// TwinCAT 3 PLC project TwinCAT3_Numpad_Keypad
// ProgramVersion: 3.1.4023.0
// libraries:
//   Tc2_Standard, * (Beckhoff Automation GmbH)
//   Tc2_System, * (Beckhoff Automation GmbH)
//   Tc3_Module, * (Beckhoff Automation GmbH)
//   VisuDialogs, * (System)
// project tree:
//   / GlobalTextList.TcGTLO, PlcTask.TcTTO, Visualization Manager.TcVMO (not stored), VISU_TASK.TcTTO
//   GVLs/ GVL.TcGVL
//   POUs/ MAIN.TcPOU
//   VISUs/Keyboard/ DialogCheckInit.TcPOU, DialogCheckInitForExponential.TcPOU, Dialog_Constants.TcGVL, Dialog_FormatTypes.TcDUT, Dialog_Variables_Exp.TcGVL, Keypad.TcVIS, KeypadLayout.TcVIS, Keypad_Original.TcVIS, Numpad.TcVIS, NumpadExtended.TcVIS, Numpad_Original.TcVIS, VisuDlg_CheckedAppend.TcPOU, VisuDlg_CheckedClear.TcPOU, VisuDlg_CheckedExpFloatFormatSwitch.TcPOU, VisuDlg_GetPasswordString.TcPOU, VisuDlg_ProcessBack.TcPOU, VisuDlg_ProcessChangeNumberFormat.TcPOU, VisuDlg_ProcessChangeSign.TcPOU, VisuDlg_ProcessChangeSignExtended.TcPOU, VisuDlg_ProcessChar.TcPOU, VisuDlg_ProcessCharWithInit.TcPOU, VisuDlg_ProcessClear.TcPOU, VisuDlg_ProcessExp.TcPOU, VisuDlg_ProcessExpFloatFormatSwitch.TcPOU
//   VISUs/ vMain.TcVIS

CONFIGURATION TwinCAT3_Numpad_Keypad
    RESOURCE PLC ON TwinCAT3
        TASK PlcTask(INTERVAL := T#10ms, PRIORITY := 20);
        TASK VISU_TASK(INTERVAL := T#1ms, PRIORITY := 30);
        PROGRAM MAIN WITH PlcTask : MAIN;
        PROGRAM VisuElems_Visu_Prg WITH VISU_TASK : VisuElems.Visu_Prg;
    END_RESOURCE
END_CONFIGURATION

// ---- VISUs/Keyboard/Dialog_FormatTypes.TcDUT
{attribute 'qualified_only'}
TYPE Dialog_FormatTypes :
(
	DECIMAL := 0,
	HEX
);
END_TYPE

// ---- GVLs/GVL.TcGVL
VAR_GLOBAL
  gsPadTitle: STRING;
END_VAR

// ---- VISUs/Keyboard/Dialog_Constants.TcGVL
{attribute 'explicit-init-exit-handling' := 'visu'}
{attribute 'qualified_only'}
VAR_GLOBAL CONSTANT
	PASSWORD_CHAR : STRING(1) := '*';
END_VAR
VAR_GLOBAL
	stTabl: INT;
END_VAR

// ---- VISUs/Keyboard/Dialog_Variables_Exp.TcGVL
{attribute 'explicit-init-exit-handling' := 'visu'}
{attribute: 'global_init_slot' := '150000'}
VAR_GLOBAL
	// Value contains e (exp was pressed)
	g_XExp : BOOL;
END_VAR

// ---- POUs/MAIN.TcPOU
PROGRAM MAIN
VAR
  nTest: INT;
  sTest: STRING;
END_VAR

END_PROGRAM

// ---- VISUs/Keyboard/DialogCheckInit.TcPOU
FUNCTION DialogCheckInit : BOOL
VAR_IN_OUT
	stValue : STRING;
	stOutput : STRING;
	bInit : BOOL;
END_VAR
VAR
END_VAR

IF bInit THEN
	stValue := ''; 
	stOutput := '';
	g_XExp := FALSE;
	// g_Format is reset on close, not on init
	bInit := FALSE;
END_IF

END_FUNCTION

// ---- VISUs/Keyboard/DialogCheckInitForExponential.TcPOU
// On opening of the NumpadExtended, we have to check the display value.
// It can be displayed in exponential notation.
// New function used with the VisuDlg_Process.. functions
FUNCTION DialogCheckInitForExponential : BOOL
VAR_IN_OUT	
	bInit : BOOL;
END_VAR
VAR_INPUT
	stValue : STRING;
END_VAR

// Starting with V3.5.9.0 the value will not be reset, after the first 
// action. Because of the new usage of the textfield with caret and selection.
IF bInit THEN
	bInit := FALSE;
	g_XExp := FALSE;
	
	IF 0 < LEN(stValue) THEN
		// value contains the 'e' character: set flag g_XExp 
		IF FIND(stValue, 'e') > 0 THEN
			g_XExp := TRUE;
		END_IF
	END_IF
	
END_IF

END_FUNCTION

// ---- VISUs/Keyboard/VisuDlg_CheckedAppend.TcPOU
FUNCTION VisuDlg_CheckedAppend : BOOL
VAR_IN_OUT
	stOutputValue : STRING;
	stVariableValue : STRING;
	bInit : BOOL;
END_VAR
VAR_INPUT
	bPassword : BOOL;
	cToAppend : STRING(1);
END_VAR

DialogCheckInit(stVariableValue, stOutputValue, bInit);

stVariableValue := CONCAT(stVariableValue, cToAppend);
IF bPassword THEN
	stOutputValue := CONCAT(stOutputValue, Dialog_Constants.PASSWORD_CHAR);
ELSE
	stOutputValue := stVariableValue;
END_IF

END_FUNCTION

// ---- VISUs/Keyboard/VisuDlg_CheckedClear.TcPOU
// clear for the Numpad, not NumpadBasic
FUNCTION VisuDlg_CheckedClear : Bool
VAR_IN_OUT
	stOutputValue : STRING;
	stVariableValue : STRING;
	flags : DWORD;
END_VAR
VAR
END_VAR

// because of integrated visu, put into a function.
// reason: unknown g_XExp
stVariableValue := '';
stOutputValue := '';
g_XExp := FALSE;
flags := flags AND NOT SINT_TO_DWORD(16#0008);
flags := flags AND NOT SINT_TO_DWORD(16#0010);

END_FUNCTION

// ---- VISUs/Keyboard/VisuDlg_CheckedExpFloatFormatSwitch.TcPOU
// switches the format of the displayed value
// between exponential and float / decimal value
FUNCTION VisuDlg_CheckedExpFloatFormatSwitch : BOOL
VAR_IN_OUT
	stOutputValue : STRING;
	stVariableValue : STRING;
END_VAR
VAR_INPUT
	bPassword: BOOL;
END_VAR
VAR
	// no need to initialize the global flag for exp
	bInitExp : BOOL := FALSE;
	// just dummies, not needed here
	iCaretPosition		: INT;
	iSelectionStart		: INT;
	iSelectionEnd		: INT;
END_VAR

//dont call DialogCheckInit here

VisuDlg_ProcessExpFloatFormatSwitch(stOutputValue, stVariableValue, iCaretPosition, iSelectionStart, iSelectionEnd, bInitExp, bPassword);

END_FUNCTION

// ---- VISUs/Keyboard/VisuDlg_ProcessExpFloatFormatSwitch.TcPOU
/// switches the format of the displayed value
/// between exponential and float / decimal value
/// and changes caret position and selection
FUNCTION VisuDlg_ProcessExpFloatFormatSwitch : BOOL
VAR_IN_OUT
	stOutputValue : STRING;
	stVariableValue : STRING;
	/// The current position of the caret. Either within the text or at the end of the text
	iCaretPosition		: INT;
	/// The start of the selected text (1-relative)
	iSelectionStart		: INT;
	/// The end of the selected text (1-relative). If the complete text is selected this
	/// parameter is textlength + 1
	iSelectionEnd		: INT;		
	/// Initialize of global value for extended numpad, should be done with the first action.
	bInit 				: BOOL;
END_VAR
VAR_INPUT
	bPassword: BOOL;
END_VAR
VAR
	rBuffer : REAL;
	/// Helper class, that formats real variables using a custom format string
	{attribute 'ieccodeconversion_datatype' := 'VisuElemBase.VisuFbPrintfRealVarConverted'}
	PrintfRealVar : VisuElems.VisuFbPrintfRealVar;
	// just defined string size
	stResult : STRING(50);	
	sFormat : STRING;
	i : INT;
END_VAR

DialogCheckInitForExponential(bInit, stVariableValue);

IF g_XExp = FALSE THEN
	g_XExp := TRUE;
	sFormat := '%e';
ELSE
	g_XExp := FALSE;
	sFormat := '%g';
END_IF

rBuffer := STRING_TO_REAL(stVariableValue);

// we always use string, and not wstring
PrintfRealVar.SetVariable(ADR(rBuffer));
PrintfRealVar.pBuffer := ADR(stResult);
PrintfRealVar.dwBufferSize := 50;
PrintfRealVar.Printf(ADR(sFormat));

stVariableValue := stResult;

IF bPassword THEN
	stOutputValue := '';
	FOR i := 0 TO LEN(stVariableValue) - 1 DO
		stOutputValue := CONCAT(stOutputValue, Dialog_Constants.PASSWORD_CHAR);
	END_FOR
ELSE
	stOutputValue := stVariableValue;
END_IF

// set the caret to the end of the value:
iCaretPosition := LEN(stOutputValue) + 1;
iSelectionStart := iSelectionEnd := iCaretPosition;

END_FUNCTION

// ---- VISUs/Keyboard/VisuDlg_GetPasswordString.TcPOU
FUNCTION VisuDlg_GetPasswordString : STRING
VAR_INPUT
	stOrg : STRING;
END_VAR
VAR
	i : INT;
	iLen : INT;
END_VAR

iLen := LEN(stOrg);
FOR i := 0 TO iLen - 1 DO
	VisuDlg_GetPasswordString := CONCAT(VisuDlg_GetPasswordString, '*');
END_FOR

END_FUNCTION

// ---- VISUs/Keyboard/VisuDlg_ProcessBack.TcPOU
/// This function processes the <back> character according to the caret position and/or the current selection.
/// Additional, values for the numpadextended will be initialised once
FUNCTION VisuDlg_ProcessBack
VAR_IN_OUT
	/// This is the string representation of the variable value, that will be displayed
	/// in the visualization. If the flag xPassword is TRUE the variable value will be
	/// display with password characters
	stOutputValue		: STRING;
	/// This parameter is the variable value, where the character is appended/inserted
	stVariableValue		: STRING;
	/// The current position of the caret. Either within the text or at the end of the text
	iCaretPosition		: INT;
	/// The start of the selected text (1-relative)
	iSelectionStart		: INT;
	/// The end of the selected text (1-relative). If the complete text is selected this
	/// parameter is textlength + 1
	iSelectionEnd		: INT;
	/// Initialize of global value, should be done with the first action.
	bInit 				: BOOL;	
END_VAR
VAR
	iTextLength			: INT;
	iPositionToDelete	: INT;
	iCountCharsToDelete	: INT;
	// Before deleting the text we store the text to delete
	sDeletedText		: STRING;
END_VAR

DialogCheckInitForExponential(bInit, stVariableValue);

// stOutputValue and stVariableValue should have the same length
iTextLength := LEN(stVariableValue);

IF 0 < iTextLength THEN
	IF iSelectionStart = iSelectionEnd THEN
		// No selection exists. We delete the character left the caret. It is necessary, that the caret is right the
		// 1st character, i.e. the caret position must be > 1
		IF iTextLength + 1 <= iCaretPosition THEN
			// Caret at the end of the text. Delete the last character
			sDeletedText := RIGHT(stVariableValue, 1);
			stVariableValue := LEFT(stVariableValue, iTextLength - 1);
			stOutputValue := LEFT(stOutputValue, iTextLength - 1);
			// The caret moves one position to the left
			iCaretPosition := iCaretPosition - 1;
		ELSIF 1 < iCaretPosition THEN
			iPositionToDelete := iCaretPosition - 1;
			sDeletedText := MID(stVariableValue, 1, iPositionToDelete);
			stVariableValue := DELETE(stVariableValue, 1, iPositionToDelete);
			stOutputValue := DELETE(stOutputValue, 1, iPositionToDelete);
			// The caret moves one position to the left
			iCaretPosition := iCaretPosition - 1;
		END_IF
	ELSE
		// The back key deletes the selected text and after that the caret is at the selection begin.
		iCaretPosition := iSelectionStart;
	
		iCountCharsToDelete := iSelectionEnd - iSelectionStart;
		sDeletedText := MID(stVariableValue, iCountCharsToDelete, iSelectionStart);
		stVariableValue := DELETE(stVariableValue, iCountCharsToDelete, iSelectionStart);
		stOutputValue := DELETE(stOutputValue, iCountCharsToDelete, iSelectionStart);
		
		// After that no selection exists.
		iSelectionEnd := iSelectionStart;
	END_IF
END_IF

IF g_XExp THEN
	// If the 'e' character was deleted, we reset the g_XExp flag 
	g_XExp := 0 = FIND(sDeletedText, 'e');
END_IF

END_FUNCTION

// ---- VISUs/Keyboard/VisuDlg_ProcessChangeNumberFormat.TcPOU
/// Update the variable display value in the Numpad for hex or dec and change the radio button.
/// This function is an enhancement of function VisuDlg_CheckedChangeNumberFormat, that also modifies
/// the caret and selection if the caret would be outside the text after the change of the display format.
/// :return: Not used, always FALSE
FUNCTION VisuDlg_ProcessChangeNumberFormat : BOOL
VAR_IN_OUT
	stOutputValue : STRING;
	stVariableValue : STRING;
	stMin : STRING;
	stMax : STRING;
	iFormatValue : INT;
	/// The current position of the caret. Either within the text or at the end of the text
	iCaretPosition	: INT;
	/// The start of the selected text (1-relative)
	iSelectionStart	: INT;
	/// The end of the selected text (1-relative).
	iSelectionEnd	: INT;
END_VAR
VAR_INPUT
	bPassword: BOOL;
	// use this way, because of integrated visu
	// 0. dec , 1. hex
	stClickedRadio : STRING;
END_VAR
VAR
	i : INT;	
	bChanged : BOOL;
	iTextLengthBeforeChange	: INT;
END_VAR

// simulate the radio button change
IF iFormatValue = Dialog_FormatTypes.HEX AND stClickedRadio = '0' THEN
	iFormatValue := Dialog_FormatTypes.DECIMAL;	
	bChanged := TRUE;
ELSIF iFormatValue = Dialog_FormatTypes.DECIMAL AND stClickedRadio = '1' THEN
	iFormatValue := Dialog_FormatTypes.HEX;
	bChanged := TRUE;
END_IF

// do some additional stuff
IF bChanged THEN
	// In order to check, whether the caret and/or selection has to be adjusted, we determine
	// the text length before the change, that corresponds to the parameters iCaretPosition and iSelection[Start|End]
	iTextLengthBeforeChange := LEN(stVariableValue);

	IF iFormatValue = Dialog_FormatTypes.HEX THEN	
		IF g_XExp THEN
			// first change the value to float:
			VisuDlg_CheckedExpFloatFormatSwitch(stOutputValue, stVariableValue, bPassword);
		END_IF
		stVariableValue := VisuDlgUtil_FormatValueToHex(stVariableValue);
		
		IF stMin <> '' THEN
			stMin := VisuDlgUtil_FormatExpToG(stMin);
		END_IF
		IF stMax <> '' THEN
			stMax := VisuDlgUtil_FormatExpToG(stMax);
		END_IF
	ELSE	
		stVariableValue := VisuDlgUtil_FormatValueToDec(stVariableValue);
		IF stMin <> '' THEN
			stMin := VisuDlgUtil_FormatValueToDec(stMin);
		END_IF
		IF stMax <> '' THEN
			stMax := VisuDlgUtil_FormatValueToDec(stMax);
		END_IF
	END_IF
	
	VisuDlgUtil_UpdateOutputValue(stOutputValue, stVariableValue, bPassword);
	
	// We adjust the caret and the selection.
	VisuDlgUtil_AdjustCaretAndSelectionAfterNumberFormatChange(
		iTextLengthBeforeChange,
		stVariableValue,
		iCaretPosition,
		iSelectionStart,
		iSelectionEnd
	);
END_IF

END_FUNCTION

// ---- VISUs/Keyboard/VisuDlg_ProcessChangeSign.TcPOU
/// This function changes the sign of the value
/// and changes caret position and selection accordingly
FUNCTION VisuDlg_ProcessChangeSign : BOOL
VAR_IN_OUT
	stOutputValue : STRING;
	stVariableValue : STRING;
	/// The current position of the caret. Either within the text or at the end of the text
	iCaretPosition		: INT;
	/// The start of the selected text (1-relative)
	iSelectionStart		: INT;
	/// The end of the selected text (1-relative). If the complete text is selected this
	/// parameter is textlength + 1
	iSelectionEnd		: INT;
END_VAR
VAR_INPUT
	bPassword: BOOL;
END_VAR
VAR
	// init only needed for numpadextended
	bInit : BOOL := FALSE;
END_VAR

VisuDlg_ProcessChangeSign := 
VisuDlg_ProcessChangeSignExtended(stOutputValue, stVariableValue, iCaretPosition, iSelectionStart, iSelectionEnd, bInit, bPassword, 0);

END_FUNCTION

// ---- VISUs/Keyboard/VisuDlg_ProcessChangeSignExtended.TcPOU
/// Replaces VisuDlg_CheckedChangeSignExtended.
/// For usage of caret and selection, we use a different init, only of the global flag exp.
FUNCTION VisuDlg_ProcessChangeSignExtended : BOOL
VAR_IN_OUT
	stOutputValue : STRING;
	stVariableValue : STRING;
	/// The current position of the caret. Either within the text or at the end of the text
	iCaretPosition		: INT;
	/// The start of the selected text (1-relative)
	iSelectionStart		: INT;
	/// The end of the selected text (1-relative). If the complete text is selected this
	/// parameter is textlength + 1
	iSelectionEnd		: INT;
	// inits only the global flag for exp.
	bInit : BOOL;
END_VAR
VAR_INPUT
	bPassword: BOOL;
	iFormatValue : INT;
END_VAR
VAR
	iPos : INT;
	iBuffer : INT;
	stBuffer : STRING;
END_VAR

DialogCheckInitForExponential(bInit, stVariableValue);

IF LEN(stVariableValue) > 0 THEN
	IF g_XExp = FALSE THEN
		// 45: -
		// change - to +, but + is not displayed
		IF stVariableValue[0] = 45 THEN
			stVariableValue := RIGHT(stVariableValue, LEN(stVariableValue) - 1);						
			IF bPassword THEN
				stOutputValue := RIGHT(stOutputValue, LEN(stOutputValue) - 1);
			END_IF
			iCaretPosition := iCaretPosition - 1;
			iSelectionStart := iSelectionStart - 1;
			iSelectionEnd := iSelectionEnd - 1;
		ELSE
			// change + to -
			IF iFormatValue = Dialog_FormatTypes.HEX THEN
				// in hex the - is never displayed, but the value is changed:
				// 2 with +/-: 		-> F..FE
				// F..FE with +/- 	-> 2				
				stBuffer := CONCAT('16#', stVariableValue);
				iBuffer := STRING_TO_INT(stBuffer);
				IF iBuffer < 0 THEN
					// F..FE with +/- 	-> 2
					iBuffer := (-1) * iBuffer;
					stBuffer := INT_TO_STRING(iBuffer);
				ELSE	
					// 2 with +/-: 		-> F..FE				
					stBuffer := CONCAT('-', INT_TO_STRING(iBuffer));
				END_IF				
			END_IF
			stVariableValue := CONCAT('-', stVariableValue);			
			IF bPassword THEN
				stOutputValue := CONCAT(stOutputValue, Dialog_Constants.PASSWORD_CHAR);
			END_IF
			IF iFormatValue = Dialog_FormatTypes.DECIMAL THEN
				iCaretPosition := iCaretPosition + 1;
				iSelectionStart := iSelectionStart + 1;
				iSelectionEnd := iSelectionEnd + 1;
			END_IF
		END_IF
		IF iFormatValue = Dialog_FormatTypes.HEX THEN
			stVariableValue := VisuDlgUtil_FormatValueToHex(stBuffer);
			// set to the end
			iCaretPosition := LEN(stVariableValue) + 1;
			iSelectionStart := iCaretPosition;
			iSelectionEnd := iCaretPosition;		
		END_IF
	ELSE
		// find the 'e' in the value and change the sign behind it.
		// with 'e' we always show a sign
		iPos := FIND(stVariableValue, 'e');
		IF iPos > 0 THEN
			IF stVariableValue[iPos] = 45 THEN
				// change - to +:
				stVariableValue := REPLACE(stVariableValue, '+', 1, iPos+1);				
			ELSE
				stVariableValue := REPLACE(stVariableValue, '-', 1, iPos+1);	
			END_IF			
		END_IF		
	END_IF
END_IF
IF NOT bPassword THEN
	stOutputValue := stVariableValue;
END_IF

END_FUNCTION

// ---- VISUs/Keyboard/VisuDlg_ProcessChar.TcPOU
/// This function takes a given character and appends/inserts it in the string representing the variable value.
/// To decide, which action has to be performed, the current caret position and the currently selected text is
/// evaluated. 
FUNCTION VisuDlg_ProcessChar
VAR_IN_OUT
	/// This is the string representation of the variable value, that will be displayed
	/// in the visualization. If the flag xPassword is TRUE the variable value will be
	/// display with password characters
	stOutputValue		: STRING;
	/// This parameter is the variable value, where the character is appended/inserted
	stVariableValue		: STRING;
	/// The current position of the caret. Either within the text or at the end of the text
	iCaretPosition		: INT;
	/// The start of the selected text (1-relative)
	iSelectionStart		: INT;
	/// The end of the selected text (1-relative). If the complete text is selected this
	/// parameter is textlength + 1
	iSelectionEnd		: INT;
END_VAR
VAR_INPUT
	/// Inidicates, whether the entered value should be readable (FALSE) or displayed with
	/// password characters
	xPassword			: BOOL;
	/// The character to append/insert
	cToConsume			: STRING(1);
END_VAR
VAR
	// the keypad calls this method, where we dont use the global flag for exp
	bInitExp : BOOL := FALSE;
END_VAR

VisuDlg_ProcessCharWithInit(stOutputValue, stVariableValue, iCaretPosition, iSelectionStart, iSelectionEnd, bInitExp, xPassword, cToConsume);

END_FUNCTION

// ---- VISUs/Keyboard/VisuDlg_ProcessCharWithInit.TcPOU
/// This function takes a given character and appends/inserts it in the string representing the variable value.
/// To decide, which action has to be performed, the current caret position and the currently selected text is
/// evaluated. 
/// Additional, values for the numpadextended will be initialised once
FUNCTION VisuDlg_ProcessCharWithInit
VAR_IN_OUT
	/// This is the string representation of the variable value, that will be displayed
	/// in the visualization. If the flag xPassword is TRUE the variable value will be
	/// display with password characters
	stOutputValue		: STRING;
	/// This parameter is the variable value, where the character is appended/inserted
	stVariableValue		: STRING;
	/// The current position of the caret. Either within the text or at the end of the text
	iCaretPosition		: INT;
	/// The start of the selected text (1-relative)
	iSelectionStart		: INT;
	/// The end of the selected text (1-relative). If the complete text is selected this
	/// parameter is textlength + 1
	iSelectionEnd		: INT;
	/// Initialize of global value, for numpadextended, should be done with the first action.
	bInit 				: BOOL;
END_VAR
VAR_INPUT
	/// Inidicates, whether the entered value should be readable (FALSE) or displayed with
	/// password characters
	xPassword			: BOOL;
	/// The character to append/insert
	cToConsume			: STRING(1);
END_VAR
VAR
	iTextLength			: INT;
	cToConsumeInOutput	: STRING(1);
	iInsertPosition		: INT;
	iCountCharsToDelete	: INT;
	// Before deleting the text we store the text to delete
	sDeletedText		: STRING;
END_VAR

DialogCheckInitForExponential(bInit, stVariableValue);

// stOutputValue and stVariableValue should have the same length
iTextLength := LEN(stVariableValue);

IF xPassword THEN
	cToConsumeInOutput := Dialog_Constants.PASSWORD_CHAR;
ELSE
	cToConsumeInOutput := cToConsume;
END_IF

IF iSelectionStart = iSelectionEnd THEN
	// No selection exists
	IF iCaretPosition <= iTextLength THEN
		// Insert the character at the caret position. The caret position is the position before the character,
		// whereas the position parameter for the INSERT call is the position after the character.  
		iInsertPosition := iCaretPosition - 1;
		stVariableValue := INSERT(stVariableValue, cToConsume, iInsertPosition);
		stOutputValue := INSERT(stOutputValue, cToConsumeInOutput, iInsertPosition);
	ELSIF iTextLength < iCaretPosition THEN
		// Append the text
		stVariableValue := CONCAT(stVariableValue, cToConsume);
		stOutputValue := CONCAT(stOutputValue, cToConsumeInOutput);
	END_IF
ELSE
	// The character replaces the selection. After that we have no selection and the caret will at the
	// beginning of the (previous) selection
	iCaretPosition := iSelectionStart;

	iCountCharsToDelete := iSelectionEnd - iSelectionStart;
	
	sDeletedText := MID(stVariableValue, iCountCharsToDelete, iSelectionStart);
	stVariableValue := DELETE(stVariableValue, iCountCharsToDelete, iSelectionStart);
	stOutputValue := DELETE(stOutputValue, iCountCharsToDelete, iSelectionStart);

	iInsertPosition := iSelectionStart - 1;
	stVariableValue := INSERT(stVariableValue, cToConsume, iInsertPosition);
	stOutputValue := INSERT(stOutputValue, cToConsumeInOutput, iInsertPosition);
END_IF

// Caret has to move one position to the right
iCaretPosition := iCaretPosition + 1;
// Entering a character always deletes the selection. So we can simply set the selection variables
// to the caret position
iSelectionStart := iCaretPosition;
iSelectionEnd := iCaretPosition;

IF g_XExp AND_THEN 0 < LEN(sDeletedText) THEN
	// If the 'e' character was deleted, we reset the g_XExp flag 
	g_XExp := 0 = FIND(sDeletedText, 'e');
END_IF

END_FUNCTION

// ---- VISUs/Keyboard/VisuDlg_ProcessClear.TcPOU
/// This function is an enhancement of function VisuDlg_CheckedClear, that also resets the caret and
/// selection.
/// :return: Not used, always FALSE
FUNCTION VisuDlg_ProcessClear : BOOL
VAR_IN_OUT
	/// This is the string representation of the variable value, that will be displayed in the visualization.
	stOutputValue	: STRING;
	/// This parameter is the variable value, that will be cleared
	stVariableValue : STRING;
	/// See VisuDlg_CheckedClear
	flags 			: DWORD;
	/// The current position of the caret. Either within the text or at the end of the text
	iCaretPosition	: INT;
	/// The start of the selected text (1-relative)
	iSelectionStart	: INT;
	/// The end of the selected text (1-relative).
	iSelectionEnd	: INT;
END_VAR

VisuDlg_CheckedClear(stOutputValue, stVariableValue, flags);

iCaretPosition	:= 1;
iSelectionStart	:= 1;
iSelectionEnd	:= 1;

END_FUNCTION

// ---- VISUs/Keyboard/VisuDlg_ProcessExp.TcPOU
/// This function add the exponential notation to the value, shown in the numpadextended
/// and changes caret position and selection
FUNCTION VisuDlg_ProcessExp : BOOL
VAR_IN_OUT
	stOutputValue : STRING;
	stVariableValue : STRING;
	/// The current position of the caret. Either within the text or at the end of the text
	iCaretPosition		: INT;
	/// The start of the selected text (1-relative)
	iSelectionStart		: INT;
	/// The end of the selected text (1-relative). If the complete text is selected this
	/// parameter is textlength + 1
	iSelectionEnd		: INT;	
	/// Initialize of global value for extended numpad, should be done with the first action.
	bInit : BOOL;
END_VAR
VAR_INPUT
	bPassword : BOOL;
END_VAR

DialogCheckInitForExponential(bInit, stVariableValue);

IF g_XExp = FALSE THEN
	g_XExp := TRUE;	
	
	IF stVariableValue = '' THEN
		VisuDlg_CheckedAppend(stOutputValue, stVariableValue, bInit, bPassword, '0');
	END_IF
	
	VisuDlg_CheckedAppend(stOutputValue, stVariableValue, bInit, bPassword, 'e');
	VisuDlg_CheckedAppend(stOutputValue, stVariableValue, bInit, bPassword, '+');
	VisuDlg_CheckedAppend(stOutputValue, stVariableValue, bInit, bPassword, '0');
	
	// set the caret to the end of the value:
	iCaretPosition := LEN(stOutputValue) + 1;
	iSelectionStart := iSelectionEnd := iCaretPosition;
END_IF

END_FUNCTION

// ---- GlobalTextList.TcGTLO
TEXTLIST GlobalTextList
  21 = '  '
  115 = '!'
  116 = '"'
  85 = '#'
  118 = '$'
  119 = '%'
  309 = '%i'
  289 = '%s'
  129 = '&'
  883 = '&i'
  86 = "'"
  122 = '('
  123 = ')'
  111 = '*'
  932 = '+'
  5 = '+/-'
  57 = ','
  588 = '-'
  4 = '.'
  121 = '/'
  6 = '0'
  7 = '1'
  8 = '2'
  9 = '3'
  10 = '4'
  11 = '5'
  12 = '6'
  13 = '7'
  14 = '8'
  15 = '9'
  59 = ':'
  58 = ';'
  41 = '<'
  124 = '='
  419 = '>'
  126 = '?'
  87 = '@'
  63 = 'a'
  64 = 'A'
  51 = 'b'
  52 = 'B'
  3 = 'Back'
  47 = 'c'
  48 = 'C'
  2 = 'Clear'
  67 = 'd'
  68 = 'D'
  379 = 'Dec'
  92 = 'e'
  93 = 'E'
  1 = 'ESC'
  22 = 'Exp'
  69 = 'f'
  70 = 'F'
  27 = 'F - E'
  71 = 'g'
  72 = 'G'
  73 = 'h'
  74 = 'H'
  382 = 'Hex'
  102 = 'i'
  103 = 'I'
  75 = 'j'
  76 = 'J'
  199 = 'k'
  78 = 'K'
  79 = 'l'
  80 = 'L'
  55 = 'm'
  56 = 'M'
  17 = 'Max:'
  1537 = 'Min:'
  53 = 'n'
  54 = 'N'
  104 = 'o'
  105 = 'O'
  0 = 'OK'
  106 = 'p'
  107 = 'P'
  88 = 'q'
  89 = 'Q'
  94 = 'r'
  894 = 'R'
  65 = 's'
  66 = 'S'
  32 = 'Shift'
  33 = 'Space'
  96 = 't'
  97 = 'T'
  100 = 'u'
  101 = 'U'
  49 = 'v'
  50 = 'V'
  90 = 'w'
  91 = 'W'
  45 = 'x'
  46 = 'X'
  43 = 'y'
  44 = 'Y'
  98 = 'z'
  99 = 'Z'
  37 = '['
  128 = '\\'
  38 = ']'
  113 = '^'
  61 = '_'
  36 = '{'
  40 = '|'
  39 = '}'
  112 = '~'
  108 = '§'
  84 = '°'
  19 = '²'
  23 = '³'
  114 = '´'
  35 = 'ä'
  81 = 'Ä'
  29 = 'ö'
  793 = 'Ö'
  82 = 'ü'
  83 = 'Ü'
  109 = 'ß'
  28 = '€'
END_TEXTLIST

// ---- VISUs/Keyboard/Keypad.TcVIS
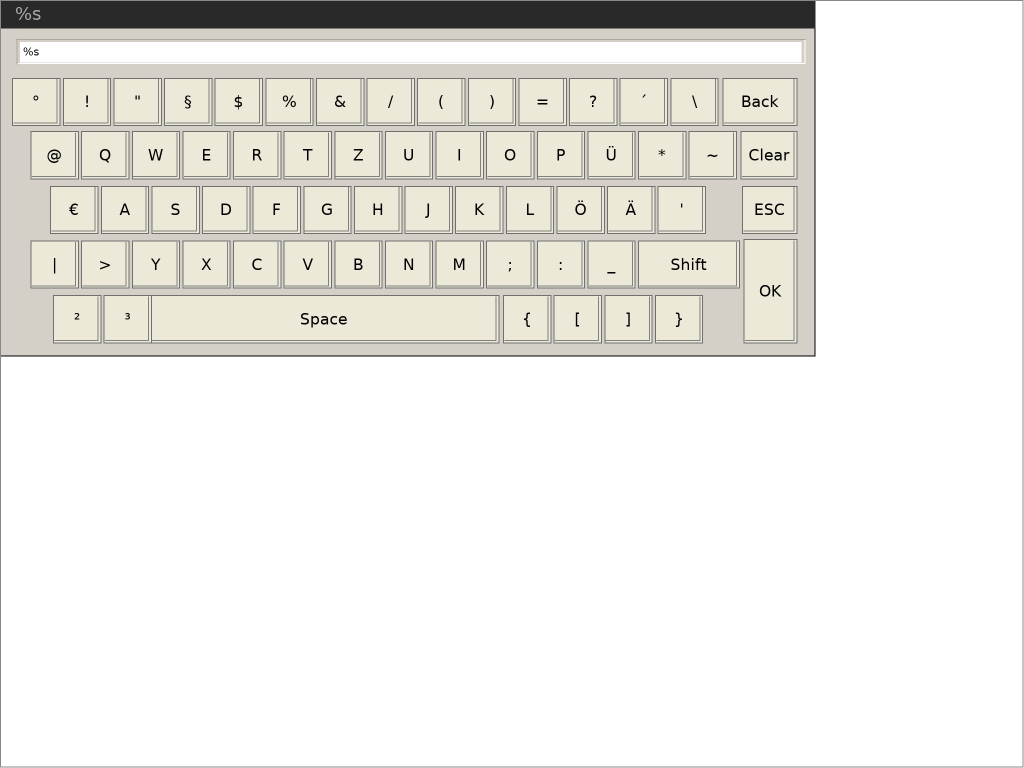
VISUALIZATION Keypad  // 1024x768
VAR_INPUT
	stVariableValue : STRING;
	stMin : STRING;
	stMax : STRING;
	wstTitle : WSTRING;
	flags : DWORD;
END_VAR
VAR
	bInit : BOOL;
	bShift : BOOL := TRUE;
	stMessage : STRING;
	stOutputValue : STRING;
	iCaretPosition	: INT;
	iSelectionStart	: INT;
	iSelectionEnd	: INT;
	xAllSelected	: BOOL;
END_VAR
    Rectangle (0,0 815x356)
    Polyline (17,64) (17,39) (805,39)
    Polyline (18,63) (805,63) (805,40)
    Textfield (20,42 781x20), "%s", text variable: stOutputValue
        p905179711: iCaretPosition
        p3815007873: iSelectionStart
        p1425650380: iSelectionEnd
        p3479897389: xAllSelected
    Rectangle (0,0 815x28), invisible if: VisuElems.g_VisualizationStyle.GetDINT('Dialog-UseHeaderColor', 0, 0) = 0
    Rectangle (12,4 793x20), "%s", text variable: gsPadTitle
    Frame (-3,71 803x275)
        shows KeypadLayout(stVariableValue := stVariableValue, bInit := bInit, bShift := bShift, stOutputValue := stOutputValue, iCaretPosition := iCaretPosition, iSelectionStart := iSelectionStart, iSelectionEnd := iSelectionEnd, flags := flags)
END_VISUALIZATION

// ---- VISUs/Keyboard/KeypadLayout.TcVIS
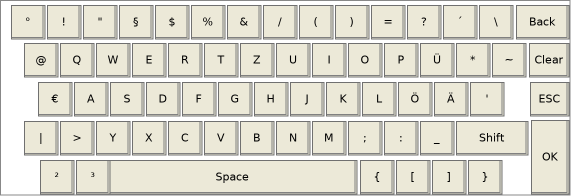
VISUALIZATION KeypadLayout  // 571x196
VAR_IN_OUT
	stVariableValue : STRING;
	bInit : BOOL;
	bShift : BOOL;
	stOutputValue : STRING;
	iCaretPosition	: INT;
	iSelectionStart	: INT;
	iSelectionEnd	: INT;
	flags: DWORD;
END_VAR
    Button (531,120 38x74), "OK"
        OnMouseDown: CloseDialog Dialog=Keypad, Result=OK, NumpadKeypad=True, NumpadKeypadSet=True
    Button (530,82 39x34), "ESC"
        OnMouseDown: CloseDialog Dialog=Keypad, Result=Cancel, NumpadKeypad=True, NumpadKeypadSet=True
    Button (529,43 40x34), "Clear"
        OnMouseDown: execute {
            stVariableValue := '';
            stOutputValue := '';
            iCaretPosition	:= 1;
            iSelectionStart	:= 1;
            iSelectionEnd := 1;
        }
    Button (516,5 53x34), "Back"
        OnMouseDown: execute { VisuDlg_ProcessBack(stOutputValue, stVariableValue, iCaretPosition, iSelectionStart, iSelectionEnd, bInit); }
    Button (456,121 72x34), "Shift"
        OnMouseDown: toggle bShift
    Button (108,160 249x34), "Space"
        OnMouseDown: execute { VisuDlg_ProcessChar(stOutputValue, stVariableValue, iCaretPosition, iSelectionStart, iSelectionEnd, (flags AND VisuElems.Visu_InputFlags.Password) = 1, ' '); }
    Button (40,160 34x34), "²"
        OnMouseDown: execute { VisuDlg_ProcessChar(stOutputValue, stVariableValue, iCaretPosition, iSelectionStart, iSelectionEnd, (flags AND VisuElems.Visu_InputFlags.Password) = 1, '²'); }
    Button (76,160 34x34), "³"
        OnMouseDown: execute { VisuDlg_ProcessChar(stOutputValue, stVariableValue, iCaretPosition, iSelectionStart, iSelectionEnd, (flags AND VisuElems.Visu_InputFlags.Password) = 1, '³'); }
    Button (360,160 34x34), "{"
        OnMouseDown: execute { VisuDlg_ProcessChar(stOutputValue, stVariableValue, iCaretPosition, iSelectionStart, iSelectionEnd, (flags AND VisuElems.Visu_InputFlags.Password) = 1, '{'); }
    Button (396,160 34x34), "["
        OnMouseDown: execute { VisuDlg_ProcessChar(stOutputValue, stVariableValue, iCaretPosition, iSelectionStart, iSelectionEnd, (flags AND VisuElems.Visu_InputFlags.Password) = 1, '['); }
    Button (432,160 34x34), "]"
        OnMouseDown: execute { VisuDlg_ProcessChar(stOutputValue, stVariableValue, iCaretPosition, iSelectionStart, iSelectionEnd, (flags AND VisuElems.Visu_InputFlags.Password) = 1, ']'); }
    Button (468,160 34x34), "}"
        OnMouseDown: execute { VisuDlg_ProcessChar(stOutputValue, stVariableValue, iCaretPosition, iSelectionStart, iSelectionEnd, (flags AND VisuElems.Visu_InputFlags.Password) = 1, '}'); }
    Button (24,121 34x34), "|"
        OnMouseDown: execute { VisuDlg_ProcessChar(stOutputValue, stVariableValue, iCaretPosition, iSelectionStart, iSelectionEnd, (flags AND VisuElems.Visu_InputFlags.Password) = 1, '|'); }
    Button (60,121 34x34), "<", invisible if: NOT bShift
        OnMouseDown: execute { VisuDlg_ProcessChar(stOutputValue, stVariableValue, iCaretPosition, iSelectionStart, iSelectionEnd, (flags AND VisuElems.Visu_InputFlags.Password) = 1, '<'); }
    Button (60,121 34x34), ">", invisible if: bShift
        OnMouseDown: execute { VisuDlg_ProcessChar(stOutputValue, stVariableValue, iCaretPosition, iSelectionStart, iSelectionEnd, (flags AND VisuElems.Visu_InputFlags.Password) = 1, '>'); }
    Button (96,121 34x34), "y", invisible if: NOT bShift
        OnMouseDown: execute { VisuDlg_ProcessChar(stOutputValue, stVariableValue, iCaretPosition, iSelectionStart, iSelectionEnd, (flags AND VisuElems.Visu_InputFlags.Password) = 1, 'y'); }
    Button (96,121 34x34), "Y", invisible if: bShift
        OnMouseDown: execute { VisuDlg_ProcessChar(stOutputValue, stVariableValue, iCaretPosition, iSelectionStart, iSelectionEnd, (flags AND VisuElems.Visu_InputFlags.Password) = 1, 'Y'); }
    Button (132,121 34x34), "x", invisible if: NOT bShift
        OnMouseDown: execute { VisuDlg_ProcessChar(stOutputValue, stVariableValue, iCaretPosition, iSelectionStart, iSelectionEnd, (flags AND VisuElems.Visu_InputFlags.Password) = 1, 'x'); }
    Button (132,121 34x34), "X", invisible if: bShift
        OnMouseDown: execute { VisuDlg_ProcessChar(stOutputValue, stVariableValue, iCaretPosition, iSelectionStart, iSelectionEnd, (flags AND VisuElems.Visu_InputFlags.Password) = 1, 'X'); }
    Button (168,121 34x34), "c", invisible if: NOT bShift
        OnMouseDown: execute { VisuDlg_ProcessChar(stOutputValue, stVariableValue, iCaretPosition, iSelectionStart, iSelectionEnd, (flags AND VisuElems.Visu_InputFlags.Password) = 1, 'c'); }
    Button (168,121 34x34), "C", invisible if: bShift
        OnMouseDown: execute { VisuDlg_ProcessChar(stOutputValue, stVariableValue, iCaretPosition, iSelectionStart, iSelectionEnd, (flags AND VisuElems.Visu_InputFlags.Password) = 1, 'C'); }
    Button (204,121 34x34), "v", invisible if: NOT bShift
        OnMouseDown: execute { VisuDlg_ProcessChar(stOutputValue, stVariableValue, iCaretPosition, iSelectionStart, iSelectionEnd, (flags AND VisuElems.Visu_InputFlags.Password) = 1, 'v'); }
    Button (204,121 34x34), "V", invisible if: bShift
        OnMouseDown: execute { VisuDlg_ProcessChar(stOutputValue, stVariableValue, iCaretPosition, iSelectionStart, iSelectionEnd, (flags AND VisuElems.Visu_InputFlags.Password) = 1, 'V'); }
    Button (240,121 34x34), "b", invisible if: NOT bShift
        OnMouseDown: execute { VisuDlg_ProcessChar(stOutputValue, stVariableValue, iCaretPosition, iSelectionStart, iSelectionEnd, (flags AND VisuElems.Visu_InputFlags.Password) = 1, 'b'); }
    Button (240,121 34x34), "B", invisible if: bShift
        OnMouseDown: execute { VisuDlg_ProcessChar(stOutputValue, stVariableValue, iCaretPosition, iSelectionStart, iSelectionEnd, (flags AND VisuElems.Visu_InputFlags.Password) = 1, 'B'); }
    Button (276,121 34x34), "n", invisible if: NOT bShift
        OnMouseDown: execute { VisuDlg_ProcessChar(stOutputValue, stVariableValue, iCaretPosition, iSelectionStart, iSelectionEnd, (flags AND VisuElems.Visu_InputFlags.Password) = 1, 'n'); }
    Button (276,121 34x34), "N", invisible if: bShift
        OnMouseDown: execute { VisuDlg_ProcessChar(stOutputValue, stVariableValue, iCaretPosition, iSelectionStart, iSelectionEnd, (flags AND VisuElems.Visu_InputFlags.Password) = 1, 'N'); }
    Button (312,121 34x34), "m", invisible if: NOT bShift
        OnMouseDown: execute { VisuDlg_ProcessChar(stOutputValue, stVariableValue, iCaretPosition, iSelectionStart, iSelectionEnd, (flags AND VisuElems.Visu_InputFlags.Password) = 1, 'm'); }
    Button (312,121 34x34), "M", invisible if: bShift
        OnMouseDown: execute { VisuDlg_ProcessChar(stOutputValue, stVariableValue, iCaretPosition, iSelectionStart, iSelectionEnd, (flags AND VisuElems.Visu_InputFlags.Password) = 1, 'M'); }
    Button (348,121 34x34), ",", invisible if: NOT bShift
        OnMouseDown: execute { VisuDlg_ProcessChar(stOutputValue, stVariableValue, iCaretPosition, iSelectionStart, iSelectionEnd, (flags AND VisuElems.Visu_InputFlags.Password) = 1, ','); }
    Button (348,121 34x34), ";", invisible if: bShift
        OnMouseDown: execute { VisuDlg_ProcessChar(stOutputValue, stVariableValue, iCaretPosition, iSelectionStart, iSelectionEnd, (flags AND VisuElems.Visu_InputFlags.Password) = 1, ';'); }
    Button (384,121 34x34), ".", invisible if: NOT bShift
        OnMouseDown: execute { VisuDlg_ProcessChar(stOutputValue, stVariableValue, iCaretPosition, iSelectionStart, iSelectionEnd, (flags AND VisuElems.Visu_InputFlags.Password) = 1, '.'); }
    Button (384,121 34x34), ":", invisible if: bShift
        OnMouseDown: execute { VisuDlg_ProcessChar(stOutputValue, stVariableValue, iCaretPosition, iSelectionStart, iSelectionEnd, (flags AND VisuElems.Visu_InputFlags.Password) = 1, ':'); }
    Button (420,121 34x34), "-", invisible if: NOT bShift
        OnMouseDown: execute { VisuDlg_ProcessChar(stOutputValue, stVariableValue, iCaretPosition, iSelectionStart, iSelectionEnd, (flags AND VisuElems.Visu_InputFlags.Password) = 1, '-'); }
    Button (420,121 34x34), "_", invisible if: bShift
        OnMouseDown: execute { VisuDlg_ProcessChar(stOutputValue, stVariableValue, iCaretPosition, iSelectionStart, iSelectionEnd, (flags AND VisuElems.Visu_InputFlags.Password) = 1, '_'); }
    Button (38,82 34x34), "€"
        OnMouseDown: execute { VisuDlg_ProcessChar(stOutputValue, stVariableValue, iCaretPosition, iSelectionStart, iSelectionEnd, (flags AND VisuElems.Visu_InputFlags.Password) = 1, '€'); }
    Button (74,82 34x34), "a", invisible if: NOT bShift
        OnMouseDown: execute { VisuDlg_ProcessChar(stOutputValue, stVariableValue, iCaretPosition, iSelectionStart, iSelectionEnd, (flags AND VisuElems.Visu_InputFlags.Password) = 1, 'a'); }
    Button (74,82 34x34), "A", invisible if: bShift
        OnMouseDown: execute { VisuDlg_ProcessChar(stOutputValue, stVariableValue, iCaretPosition, iSelectionStart, iSelectionEnd, (flags AND VisuElems.Visu_InputFlags.Password) = 1, 'A'); }
    Button (110,82 34x34), "s", invisible if: NOT bShift
        OnMouseDown: execute { VisuDlg_ProcessChar(stOutputValue, stVariableValue, iCaretPosition, iSelectionStart, iSelectionEnd, (flags AND VisuElems.Visu_InputFlags.Password) = 1, 's'); }
    Button (110,82 34x34), "S", invisible if: bShift
        OnMouseDown: execute { VisuDlg_ProcessChar(stOutputValue, stVariableValue, iCaretPosition, iSelectionStart, iSelectionEnd, (flags AND VisuElems.Visu_InputFlags.Password) = 1, 'S'); }
    Button (146,82 34x34), "d", invisible if: NOT bShift
        OnMouseDown: execute { VisuDlg_ProcessChar(stOutputValue, stVariableValue, iCaretPosition, iSelectionStart, iSelectionEnd, (flags AND VisuElems.Visu_InputFlags.Password) = 1, 'd'); }
    Button (146,82 34x34), "D", invisible if: bShift
        OnMouseDown: execute { VisuDlg_ProcessChar(stOutputValue, stVariableValue, iCaretPosition, iSelectionStart, iSelectionEnd, (flags AND VisuElems.Visu_InputFlags.Password) = 1, 'D'); }
    Button (182,82 34x34), "f", invisible if: NOT bShift
        OnMouseDown: execute { VisuDlg_ProcessChar(stOutputValue, stVariableValue, iCaretPosition, iSelectionStart, iSelectionEnd, (flags AND VisuElems.Visu_InputFlags.Password) = 1, 'f'); }
    Button (182,82 34x34), "F", invisible if: bShift
        OnMouseDown: execute { VisuDlg_ProcessChar(stOutputValue, stVariableValue, iCaretPosition, iSelectionStart, iSelectionEnd, (flags AND VisuElems.Visu_InputFlags.Password) = 1, 'F'); }
    Button (218,82 34x34), "g", invisible if: NOT bShift
        OnMouseDown: execute { VisuDlg_ProcessChar(stOutputValue, stVariableValue, iCaretPosition, iSelectionStart, iSelectionEnd, (flags AND VisuElems.Visu_InputFlags.Password) = 1, 'g'); }
    Button (218,82 34x34), "G", invisible if: bShift
        OnMouseDown: execute { VisuDlg_ProcessChar(stOutputValue, stVariableValue, iCaretPosition, iSelectionStart, iSelectionEnd, (flags AND VisuElems.Visu_InputFlags.Password) = 1, 'G'); }
    Button (254,82 34x34), "h", invisible if: NOT bShift
        OnMouseDown: execute { VisuDlg_ProcessChar(stOutputValue, stVariableValue, iCaretPosition, iSelectionStart, iSelectionEnd, (flags AND VisuElems.Visu_InputFlags.Password) = 1, 'h'); }
    Button (254,82 34x34), "H", invisible if: bShift
        OnMouseDown: execute { VisuDlg_ProcessChar(stOutputValue, stVariableValue, iCaretPosition, iSelectionStart, iSelectionEnd, (flags AND VisuElems.Visu_InputFlags.Password) = 1, 'H'); }
    Button (290,82 34x34), "j", invisible if: NOT bShift
        OnMouseDown: execute { VisuDlg_ProcessChar(stOutputValue, stVariableValue, iCaretPosition, iSelectionStart, iSelectionEnd, (flags AND VisuElems.Visu_InputFlags.Password) = 1, 'j'); }
    Button (290,82 34x34), "J", invisible if: bShift
        OnMouseDown: execute { VisuDlg_ProcessChar(stOutputValue, stVariableValue, iCaretPosition, iSelectionStart, iSelectionEnd, (flags AND VisuElems.Visu_InputFlags.Password) = 1, 'J'); }
    Button (326,82 34x34), "k", invisible if: NOT bShift
        OnMouseDown: execute { VisuDlg_ProcessChar(stOutputValue, stVariableValue, iCaretPosition, iSelectionStart, iSelectionEnd, (flags AND VisuElems.Visu_InputFlags.Password) = 1, 'k'); }
    Button (326,82 34x34), "K", invisible if: bShift
        OnMouseDown: execute { VisuDlg_ProcessChar(stOutputValue, stVariableValue, iCaretPosition, iSelectionStart, iSelectionEnd, (flags AND VisuElems.Visu_InputFlags.Password) = 1, 'K'); }
    Button (362,82 34x34), "l", invisible if: NOT bShift
        OnMouseDown: execute { VisuDlg_ProcessChar(stOutputValue, stVariableValue, iCaretPosition, iSelectionStart, iSelectionEnd, (flags AND VisuElems.Visu_InputFlags.Password) = 1, 'l'); }
    Button (362,82 34x34), "L", invisible if: bShift
        OnMouseDown: execute { VisuDlg_ProcessChar(stOutputValue, stVariableValue, iCaretPosition, iSelectionStart, iSelectionEnd, (flags AND VisuElems.Visu_InputFlags.Password) = 1, 'L'); }
    Button (398,82 34x34), "ö", invisible if: NOT bShift
        OnMouseDown: execute { VisuDlg_ProcessChar(stOutputValue, stVariableValue, iCaretPosition, iSelectionStart, iSelectionEnd, (flags AND VisuElems.Visu_InputFlags.Password) = 1, 'ö'); }
    Button (398,82 34x34), "Ö", invisible if: bShift
        OnMouseDown: execute { VisuDlg_ProcessChar(stOutputValue, stVariableValue, iCaretPosition, iSelectionStart, iSelectionEnd, (flags AND VisuElems.Visu_InputFlags.Password) = 1, 'Ö'); }
    Button (434,82 34x34), "ä", invisible if: NOT bShift
        OnMouseDown: execute { VisuDlg_ProcessChar(stOutputValue, stVariableValue, iCaretPosition, iSelectionStart, iSelectionEnd, (flags AND VisuElems.Visu_InputFlags.Password) = 1, 'ä'); }
    Button (434,82 34x34), "Ä", invisible if: bShift
        OnMouseDown: execute { VisuDlg_ProcessChar(stOutputValue, stVariableValue, iCaretPosition, iSelectionStart, iSelectionEnd, (flags AND VisuElems.Visu_InputFlags.Password) = 1, 'Ä'); }
    Button (470,82 34x34), "#", invisible if: NOT bShift
        OnMouseDown: execute { VisuDlg_ProcessChar(stOutputValue, stVariableValue, iCaretPosition, iSelectionStart, iSelectionEnd, (flags AND VisuElems.Visu_InputFlags.Password) = 1, '#'); }
    Button (470,82 34x34), "'", invisible if: bShift
        OnMouseDown: execute { VisuDlg_ProcessChar(stOutputValue, stVariableValue, iCaretPosition, iSelectionStart, iSelectionEnd, (flags AND VisuElems.Visu_InputFlags.Password) = 1, '$''); }
    Button (24,43 34x34), "@"
        OnMouseDown: execute { VisuDlg_ProcessChar(stOutputValue, stVariableValue, iCaretPosition, iSelectionStart, iSelectionEnd, (flags AND VisuElems.Visu_InputFlags.Password) = 1, '@'); }
    Button (60,43 34x34), "q", invisible if: NOT bShift
        OnMouseDown: execute { VisuDlg_ProcessChar(stOutputValue, stVariableValue, iCaretPosition, iSelectionStart, iSelectionEnd, (flags AND VisuElems.Visu_InputFlags.Password) = 1, 'q'); }
    Button (60,43 34x34), "Q", invisible if: bShift
        OnMouseDown: execute { VisuDlg_ProcessChar(stOutputValue, stVariableValue, iCaretPosition, iSelectionStart, iSelectionEnd, (flags AND VisuElems.Visu_InputFlags.Password) = 1, 'Q'); }
    Button (96,43 34x34), "w", invisible if: NOT bShift
        OnMouseDown: execute { VisuDlg_ProcessChar(stOutputValue, stVariableValue, iCaretPosition, iSelectionStart, iSelectionEnd, (flags AND VisuElems.Visu_InputFlags.Password) = 1, 'w'); }
    Button (96,43 34x34), "W", invisible if: bShift
        OnMouseDown: execute { VisuDlg_ProcessChar(stOutputValue, stVariableValue, iCaretPosition, iSelectionStart, iSelectionEnd, (flags AND VisuElems.Visu_InputFlags.Password) = 1, 'W'); }
    Button (132,43 34x34), "e", invisible if: NOT bShift
        OnMouseDown: execute { VisuDlg_ProcessChar(stOutputValue, stVariableValue, iCaretPosition, iSelectionStart, iSelectionEnd, (flags AND VisuElems.Visu_InputFlags.Password) = 1, 'e'); }
    Button (132,43 34x34), "E", invisible if: bShift
        OnMouseDown: execute { VisuDlg_ProcessChar(stOutputValue, stVariableValue, iCaretPosition, iSelectionStart, iSelectionEnd, (flags AND VisuElems.Visu_InputFlags.Password) = 1, 'E'); }
    Button (168,43 34x34), "r", invisible if: NOT bShift
        OnMouseDown: execute { VisuDlg_ProcessChar(stOutputValue, stVariableValue, iCaretPosition, iSelectionStart, iSelectionEnd, (flags AND VisuElems.Visu_InputFlags.Password) = 1, 'r'); }
    Button (168,43 34x34), "R", invisible if: bShift
        OnMouseDown: execute { VisuDlg_ProcessChar(stOutputValue, stVariableValue, iCaretPosition, iSelectionStart, iSelectionEnd, (flags AND VisuElems.Visu_InputFlags.Password) = 1, 'R'); }
    Button (204,43 34x34), "t", invisible if: NOT bShift
        OnMouseDown: execute { VisuDlg_ProcessChar(stOutputValue, stVariableValue, iCaretPosition, iSelectionStart, iSelectionEnd, (flags AND VisuElems.Visu_InputFlags.Password) = 1, 't'); }
    Button (204,43 34x34), "T", invisible if: bShift
        OnMouseDown: execute { VisuDlg_ProcessChar(stOutputValue, stVariableValue, iCaretPosition, iSelectionStart, iSelectionEnd, (flags AND VisuElems.Visu_InputFlags.Password) = 1, 'T'); }
    Button (240,43 34x34), "z", invisible if: NOT bShift
        OnMouseDown: execute { VisuDlg_ProcessChar(stOutputValue, stVariableValue, iCaretPosition, iSelectionStart, iSelectionEnd, (flags AND VisuElems.Visu_InputFlags.Password) = 1, 'z'); }
    Button (240,43 34x34), "Z", invisible if: bShift
        OnMouseDown: execute { VisuDlg_ProcessChar(stOutputValue, stVariableValue, iCaretPosition, iSelectionStart, iSelectionEnd, (flags AND VisuElems.Visu_InputFlags.Password) = 1, 'Z'); }
    Button (276,43 34x34), "u", invisible if: NOT bShift
        OnMouseDown: execute { VisuDlg_ProcessChar(stOutputValue, stVariableValue, iCaretPosition, iSelectionStart, iSelectionEnd, (flags AND VisuElems.Visu_InputFlags.Password) = 1, 'u'); }
    Button (276,43 34x34), "U", invisible if: bShift
        OnMouseDown: execute { VisuDlg_ProcessChar(stOutputValue, stVariableValue, iCaretPosition, iSelectionStart, iSelectionEnd, (flags AND VisuElems.Visu_InputFlags.Password) = 1, 'U'); }
    Button (312,43 34x34), "i", invisible if: NOT bShift
        OnMouseDown: execute { VisuDlg_ProcessChar(stOutputValue, stVariableValue, iCaretPosition, iSelectionStart, iSelectionEnd, (flags AND VisuElems.Visu_InputFlags.Password) = 1, 'i'); }
    Button (312,43 34x34), "I", invisible if: bShift
        OnMouseDown: execute { VisuDlg_ProcessChar(stOutputValue, stVariableValue, iCaretPosition, iSelectionStart, iSelectionEnd, (flags AND VisuElems.Visu_InputFlags.Password) = 1, 'I'); }
    Button (348,43 34x34), "o", invisible if: NOT bShift
        OnMouseDown: execute { VisuDlg_ProcessChar(stOutputValue, stVariableValue, iCaretPosition, iSelectionStart, iSelectionEnd, (flags AND VisuElems.Visu_InputFlags.Password) = 1, 'o'); }
    Button (348,43 34x34), "O", invisible if: bShift
        OnMouseDown: execute { VisuDlg_ProcessChar(stOutputValue, stVariableValue, iCaretPosition, iSelectionStart, iSelectionEnd, (flags AND VisuElems.Visu_InputFlags.Password) = 1, 'O'); }
    Button (384,43 34x34), "p", invisible if: NOT bShift
        OnMouseDown: execute { VisuDlg_ProcessChar(stOutputValue, stVariableValue, iCaretPosition, iSelectionStart, iSelectionEnd, (flags AND VisuElems.Visu_InputFlags.Password) = 1, 'p'); }
    Button (384,43 34x34), "P", invisible if: bShift
        OnMouseDown: execute { VisuDlg_ProcessChar(stOutputValue, stVariableValue, iCaretPosition, iSelectionStart, iSelectionEnd, (flags AND VisuElems.Visu_InputFlags.Password) = 1, 'P'); }
    Button (420,43 34x34), "ü", invisible if: NOT bShift
        OnMouseDown: execute { VisuDlg_ProcessChar(stOutputValue, stVariableValue, iCaretPosition, iSelectionStart, iSelectionEnd, (flags AND VisuElems.Visu_InputFlags.Password) = 1, 'ü'); }
    Button (420,43 34x34), "Ü", invisible if: bShift
        OnMouseDown: execute { VisuDlg_ProcessChar(stOutputValue, stVariableValue, iCaretPosition, iSelectionStart, iSelectionEnd, (flags AND VisuElems.Visu_InputFlags.Password) = 1, 'Ü'); }
    Button (456,43 34x34), "+", invisible if: NOT bShift
        OnMouseDown: execute { VisuDlg_ProcessChar(stOutputValue, stVariableValue, iCaretPosition, iSelectionStart, iSelectionEnd, (flags AND VisuElems.Visu_InputFlags.Password) = 1, '+'); }
    Button (456,43 34x34), "*", invisible if: bShift
        OnMouseDown: execute { VisuDlg_ProcessChar(stOutputValue, stVariableValue, iCaretPosition, iSelectionStart, iSelectionEnd, (flags AND VisuElems.Visu_InputFlags.Password) = 1, '*'); }
    Button (492,43 34x34), "~"
        OnMouseDown: execute { VisuDlg_ProcessChar(stOutputValue, stVariableValue, iCaretPosition, iSelectionStart, iSelectionEnd, (flags AND VisuElems.Visu_InputFlags.Password) = 1, '~'); }
    Button (11,5 34x34), "^", invisible if: NOT bShift
        OnMouseDown: execute { VisuDlg_ProcessChar(stOutputValue, stVariableValue, iCaretPosition, iSelectionStart, iSelectionEnd, (flags AND VisuElems.Visu_InputFlags.Password) = 1, '^'); }
    Button (11,5 34x34), "°", invisible if: bShift
        OnMouseDown: execute { VisuDlg_ProcessChar(stOutputValue, stVariableValue, iCaretPosition, iSelectionStart, iSelectionEnd, (flags AND VisuElems.Visu_InputFlags.Password) = 1, '°'); }
    Button (47,5 34x34), "1", invisible if: NOT bShift
        OnMouseDown: execute { VisuDlg_ProcessChar(stOutputValue, stVariableValue, iCaretPosition, iSelectionStart, iSelectionEnd, (flags AND VisuElems.Visu_InputFlags.Password) = 1, '1'); }
    Button (47,5 34x34), "!", invisible if: bShift
        OnMouseDown: execute { VisuDlg_ProcessChar(stOutputValue, stVariableValue, iCaretPosition, iSelectionStart, iSelectionEnd, (flags AND VisuElems.Visu_InputFlags.Password) = 1, '!'); }
    Button (83,5 34x34), "2", invisible if: NOT bShift
        OnMouseDown: execute { VisuDlg_ProcessChar(stOutputValue, stVariableValue, iCaretPosition, iSelectionStart, iSelectionEnd, (flags AND VisuElems.Visu_InputFlags.Password) = 1, '2'); }
    Button (83,5 34x34), """, invisible if: bShift
        OnMouseDown: execute { VisuDlg_ProcessChar(stOutputValue, stVariableValue, iCaretPosition, iSelectionStart, iSelectionEnd, (flags AND VisuElems.Visu_InputFlags.Password) = 1, '"'); }
    Button (119,5 34x34), "3", invisible if: NOT bShift
        OnMouseDown: execute { VisuDlg_ProcessChar(stOutputValue, stVariableValue, iCaretPosition, iSelectionStart, iSelectionEnd, (flags AND VisuElems.Visu_InputFlags.Password) = 1, '3'); }
    Button (119,5 34x34), "§", invisible if: bShift
        OnMouseDown: execute { VisuDlg_ProcessChar(stOutputValue, stVariableValue, iCaretPosition, iSelectionStart, iSelectionEnd, (flags AND VisuElems.Visu_InputFlags.Password) = 1, '§'); }
    Button (155,5 34x34), "4", invisible if: NOT bShift
        OnMouseDown: execute { VisuDlg_ProcessChar(stOutputValue, stVariableValue, iCaretPosition, iSelectionStart, iSelectionEnd, (flags AND VisuElems.Visu_InputFlags.Password) = 1, '4'); }
    Button (155,5 34x34), "$", invisible if: bShift
        OnMouseDown: execute { VisuDlg_ProcessChar(stOutputValue, stVariableValue, iCaretPosition, iSelectionStart, iSelectionEnd, (flags AND VisuElems.Visu_InputFlags.Password) = 1, '$$'); }
    Button (191,5 34x34), "5", invisible if: NOT bShift
        OnMouseDown: execute { VisuDlg_ProcessChar(stOutputValue, stVariableValue, iCaretPosition, iSelectionStart, iSelectionEnd, (flags AND VisuElems.Visu_InputFlags.Password) = 1, '5'); }
    Button (191,5 34x34), "%", invisible if: bShift
        OnMouseDown: execute { VisuDlg_ProcessChar(stOutputValue, stVariableValue, iCaretPosition, iSelectionStart, iSelectionEnd, (flags AND VisuElems.Visu_InputFlags.Password) = 1, '%'); }
    Button (227,5 34x34), "6", invisible if: NOT bShift
        OnMouseDown: execute { VisuDlg_ProcessChar(stOutputValue, stVariableValue, iCaretPosition, iSelectionStart, iSelectionEnd, (flags AND VisuElems.Visu_InputFlags.Password) = 1, '6'); }
    Button (227,5 34x34), "&", invisible if: bShift
        OnMouseDown: execute { VisuDlg_ProcessChar(stOutputValue, stVariableValue, iCaretPosition, iSelectionStart, iSelectionEnd, (flags AND VisuElems.Visu_InputFlags.Password) = 1, '&'); }
    Button (263,5 34x34), "7", invisible if: NOT bShift
        OnMouseDown: execute { VisuDlg_ProcessChar(stOutputValue, stVariableValue, iCaretPosition, iSelectionStart, iSelectionEnd, (flags AND VisuElems.Visu_InputFlags.Password) = 1, '7'); }
    Button (263,5 34x34), "/", invisible if: bShift
        OnMouseDown: execute { VisuDlg_ProcessChar(stOutputValue, stVariableValue, iCaretPosition, iSelectionStart, iSelectionEnd, (flags AND VisuElems.Visu_InputFlags.Password) = 1, '/'); }
    Button (299,5 34x34), "8", invisible if: NOT bShift
        OnMouseDown: execute { VisuDlg_ProcessChar(stOutputValue, stVariableValue, iCaretPosition, iSelectionStart, iSelectionEnd, (flags AND VisuElems.Visu_InputFlags.Password) = 1, '8'); }
    Button (299,5 34x34), "(", invisible if: bShift
        OnMouseDown: execute { VisuDlg_ProcessChar(stOutputValue, stVariableValue, iCaretPosition, iSelectionStart, iSelectionEnd, (flags AND VisuElems.Visu_InputFlags.Password) = 1, '('); }
    Button (335,5 34x34), "9", invisible if: NOT bShift
        OnMouseDown: execute { VisuDlg_ProcessChar(stOutputValue, stVariableValue, iCaretPosition, iSelectionStart, iSelectionEnd, (flags AND VisuElems.Visu_InputFlags.Password) = 1, '9'); }
    Button (335,5 34x34), ")", invisible if: bShift
        OnMouseDown: execute { VisuDlg_ProcessChar(stOutputValue, stVariableValue, iCaretPosition, iSelectionStart, iSelectionEnd, (flags AND VisuElems.Visu_InputFlags.Password) = 1, ')'); }
    Button (371,5 34x34), "0", invisible if: NOT bShift
        OnMouseDown: execute { VisuDlg_ProcessChar(stOutputValue, stVariableValue, iCaretPosition, iSelectionStart, iSelectionEnd, (flags AND VisuElems.Visu_InputFlags.Password) = 1, '0'); }
    Button (371,5 34x34), "=", invisible if: bShift
        OnMouseDown: execute { VisuDlg_ProcessChar(stOutputValue, stVariableValue, iCaretPosition, iSelectionStart, iSelectionEnd, (flags AND VisuElems.Visu_InputFlags.Password) = 1, '='); }
    Button (407,5 34x34), "ß", invisible if: NOT bShift
        OnMouseDown: execute { VisuDlg_ProcessChar(stOutputValue, stVariableValue, iCaretPosition, iSelectionStart, iSelectionEnd, (flags AND VisuElems.Visu_InputFlags.Password) = 1, 'ß'); }
    Button (407,5 34x34), "?", invisible if: bShift
        OnMouseDown: execute { VisuDlg_ProcessChar(stOutputValue, stVariableValue, iCaretPosition, iSelectionStart, iSelectionEnd, (flags AND VisuElems.Visu_InputFlags.Password) = 1, '?'); }
    Button (443,5 34x34), "´"
        OnMouseDown: execute { VisuDlg_ProcessChar(stOutputValue, stVariableValue, iCaretPosition, iSelectionStart, iSelectionEnd, (flags AND VisuElems.Visu_InputFlags.Password) = 1, '´'); }
    Button (479,5 34x34), "\"
        OnMouseDown: execute { VisuDlg_ProcessChar(stOutputValue, stVariableValue, iCaretPosition, iSelectionStart, iSelectionEnd, (flags AND VisuElems.Visu_InputFlags.Password) = 1, '\'); }
END_VISUALIZATION

// ---- VISUs/Keyboard/Keypad_Original.TcVIS
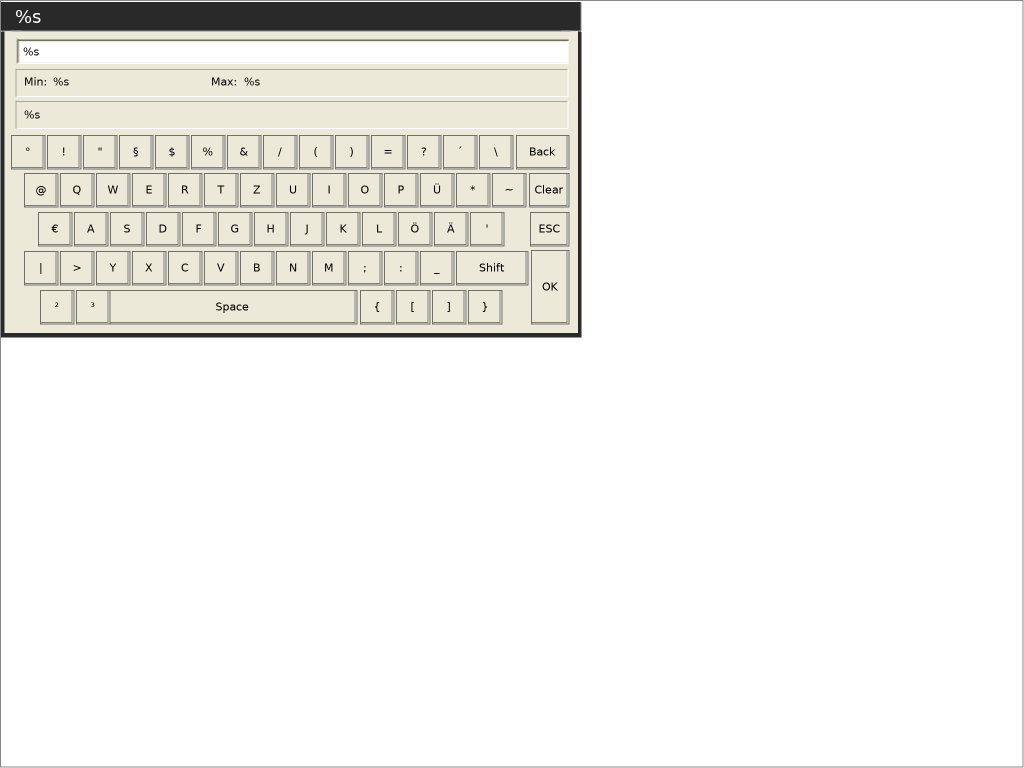
VISUALIZATION Keypad_Original  // 1024x768
VAR_INPUT
	stVariableValue : STRING;
	stMin : STRING;
	stMax : STRING;
	wstTitle : WSTRING;
	flags : DWORD;
END_VAR
VAR
	bInit : BOOL;
	bShift : BOOL := TRUE;
	stMessage : STRING;
	stOutputValue : STRING;
	iCaretPosition	: INT;
	iSelectionStart	: INT;
	iSelectionEnd	: INT;
	xAllSelected	: BOOL;
END_VAR
    Rectangle (2,28 578x40)
    Polyline (17,63) (17,39) (568,39)
    Polyline (18,63) (568,63) (568,40)
    Polyline (18,62) (18,40) (568,40)
    Textfield (20,42 547x20), "%s", text variable: stOutputValue
        p905179711: iCaretPosition
        p3815007873: iSelectionStart
        p1425650380: iSelectionEnd
        p3479897389: xAllSelected
    Rectangle (2,128 578x55)
    Rectangle (2,172 578x40)
    Rectangle (2,211 578x40)
    Rectangle (2,250 578x39)
    Rectangle (2,287 578x48)
    Button (531,250 38x74), "OK"
        OnMouseDown: CloseDialog Dialog=Keypad, Result=OK, NumpadKeypad=True, NumpadKeypadSet=True
    Button (530,212 39x34), "ESC"
        OnMouseDown: CloseDialog Dialog=Keypad, Result=Cancel, NumpadKeypad=True, NumpadKeypadSet=True
    Button (529,173 40x34), "Clear"
        OnMouseDown: execute {
            stVariableValue := '';
            stOutputValue := '';
            iCaretPosition	:= 1;
            iSelectionStart	:= 1;
            iSelectionEnd := 1;
        }
    Button (516,135 53x34), "Back"
        OnMouseDown: execute { VisuDlg_ProcessBack(stOutputValue, stVariableValue, iCaretPosition, iSelectionStart, iSelectionEnd, bInit); }
    Button (456,251 72x34), "Shift"
        OnMouseDown: toggle bShift
    Button (108,290 249x34), "Space"
        OnMouseDown: execute { VisuDlg_ProcessChar(stOutputValue, stVariableValue, iCaretPosition, iSelectionStart, iSelectionEnd, (flags AND VisuElems.Visu_InputFlags.Password) = 1, ' '); }
    Button (40,290 34x34), "²"
        OnMouseDown: execute { VisuDlg_ProcessChar(stOutputValue, stVariableValue, iCaretPosition, iSelectionStart, iSelectionEnd, (flags AND VisuElems.Visu_InputFlags.Password) = 1, '²'); }
    Button (76,290 34x34), "³"
        OnMouseDown: execute { VisuDlg_ProcessChar(stOutputValue, stVariableValue, iCaretPosition, iSelectionStart, iSelectionEnd, (flags AND VisuElems.Visu_InputFlags.Password) = 1, '³'); }
    Button (360,290 34x34), "{"
        OnMouseDown: execute { VisuDlg_ProcessChar(stOutputValue, stVariableValue, iCaretPosition, iSelectionStart, iSelectionEnd, (flags AND VisuElems.Visu_InputFlags.Password) = 1, '{'); }
    Button (396,290 34x34), "["
        OnMouseDown: execute { VisuDlg_ProcessChar(stOutputValue, stVariableValue, iCaretPosition, iSelectionStart, iSelectionEnd, (flags AND VisuElems.Visu_InputFlags.Password) = 1, '['); }
    Button (432,290 34x34), "]"
        OnMouseDown: execute { VisuDlg_ProcessChar(stOutputValue, stVariableValue, iCaretPosition, iSelectionStart, iSelectionEnd, (flags AND VisuElems.Visu_InputFlags.Password) = 1, ']'); }
    Button (468,290 34x34), "}"
        OnMouseDown: execute { VisuDlg_ProcessChar(stOutputValue, stVariableValue, iCaretPosition, iSelectionStart, iSelectionEnd, (flags AND VisuElems.Visu_InputFlags.Password) = 1, '}'); }
    Button (24,251 34x34), "|"
        OnMouseDown: execute { VisuDlg_ProcessChar(stOutputValue, stVariableValue, iCaretPosition, iSelectionStart, iSelectionEnd, (flags AND VisuElems.Visu_InputFlags.Password) = 1, '|'); }
    Button (60,251 34x34), "<", invisible if: NOT bShift
        OnMouseDown: execute { VisuDlg_ProcessChar(stOutputValue, stVariableValue, iCaretPosition, iSelectionStart, iSelectionEnd, (flags AND VisuElems.Visu_InputFlags.Password) = 1, '<'); }
    Button (60,251 34x34), ">", invisible if: bShift
        OnMouseDown: execute { VisuDlg_ProcessChar(stOutputValue, stVariableValue, iCaretPosition, iSelectionStart, iSelectionEnd, (flags AND VisuElems.Visu_InputFlags.Password) = 1, '>'); }
    Button (96,251 34x34), "y", invisible if: NOT bShift
        OnMouseDown: execute { VisuDlg_ProcessChar(stOutputValue, stVariableValue, iCaretPosition, iSelectionStart, iSelectionEnd, (flags AND VisuElems.Visu_InputFlags.Password) = 1, 'y'); }
    Button (96,251 34x34), "Y", invisible if: bShift
        OnMouseDown: execute { VisuDlg_ProcessChar(stOutputValue, stVariableValue, iCaretPosition, iSelectionStart, iSelectionEnd, (flags AND VisuElems.Visu_InputFlags.Password) = 1, 'Y'); }
    Button (132,251 34x34), "x", invisible if: NOT bShift
        OnMouseDown: execute { VisuDlg_ProcessChar(stOutputValue, stVariableValue, iCaretPosition, iSelectionStart, iSelectionEnd, (flags AND VisuElems.Visu_InputFlags.Password) = 1, 'x'); }
    Button (132,251 34x34), "X", invisible if: bShift
        OnMouseDown: execute { VisuDlg_ProcessChar(stOutputValue, stVariableValue, iCaretPosition, iSelectionStart, iSelectionEnd, (flags AND VisuElems.Visu_InputFlags.Password) = 1, 'X'); }
    Button (168,251 34x34), "c", invisible if: NOT bShift
        OnMouseDown: execute { VisuDlg_ProcessChar(stOutputValue, stVariableValue, iCaretPosition, iSelectionStart, iSelectionEnd, (flags AND VisuElems.Visu_InputFlags.Password) = 1, 'c'); }
    Button (168,251 34x34), "C", invisible if: bShift
        OnMouseDown: execute { VisuDlg_ProcessChar(stOutputValue, stVariableValue, iCaretPosition, iSelectionStart, iSelectionEnd, (flags AND VisuElems.Visu_InputFlags.Password) = 1, 'C'); }
    Button (204,251 34x34), "v", invisible if: NOT bShift
        OnMouseDown: execute { VisuDlg_ProcessChar(stOutputValue, stVariableValue, iCaretPosition, iSelectionStart, iSelectionEnd, (flags AND VisuElems.Visu_InputFlags.Password) = 1, 'v'); }
    Button (204,251 34x34), "V", invisible if: bShift
        OnMouseDown: execute { VisuDlg_ProcessChar(stOutputValue, stVariableValue, iCaretPosition, iSelectionStart, iSelectionEnd, (flags AND VisuElems.Visu_InputFlags.Password) = 1, 'V'); }
    Button (240,251 34x34), "b", invisible if: NOT bShift
        OnMouseDown: execute { VisuDlg_ProcessChar(stOutputValue, stVariableValue, iCaretPosition, iSelectionStart, iSelectionEnd, (flags AND VisuElems.Visu_InputFlags.Password) = 1, 'b'); }
    Button (240,251 34x34), "B", invisible if: bShift
        OnMouseDown: execute { VisuDlg_ProcessChar(stOutputValue, stVariableValue, iCaretPosition, iSelectionStart, iSelectionEnd, (flags AND VisuElems.Visu_InputFlags.Password) = 1, 'B'); }
    Button (276,251 34x34), "n", invisible if: NOT bShift
        OnMouseDown: execute { VisuDlg_ProcessChar(stOutputValue, stVariableValue, iCaretPosition, iSelectionStart, iSelectionEnd, (flags AND VisuElems.Visu_InputFlags.Password) = 1, 'n'); }
    Button (276,251 34x34), "N", invisible if: bShift
        OnMouseDown: execute { VisuDlg_ProcessChar(stOutputValue, stVariableValue, iCaretPosition, iSelectionStart, iSelectionEnd, (flags AND VisuElems.Visu_InputFlags.Password) = 1, 'N'); }
    Button (312,251 34x34), "m", invisible if: NOT bShift
        OnMouseDown: execute { VisuDlg_ProcessChar(stOutputValue, stVariableValue, iCaretPosition, iSelectionStart, iSelectionEnd, (flags AND VisuElems.Visu_InputFlags.Password) = 1, 'm'); }
    Button (312,251 34x34), "M", invisible if: bShift
        OnMouseDown: execute { VisuDlg_ProcessChar(stOutputValue, stVariableValue, iCaretPosition, iSelectionStart, iSelectionEnd, (flags AND VisuElems.Visu_InputFlags.Password) = 1, 'M'); }
    Button (348,251 34x34), ",", invisible if: NOT bShift
        OnMouseDown: execute { VisuDlg_ProcessChar(stOutputValue, stVariableValue, iCaretPosition, iSelectionStart, iSelectionEnd, (flags AND VisuElems.Visu_InputFlags.Password) = 1, ','); }
    Button (348,251 34x34), ";", invisible if: bShift
        OnMouseDown: execute { VisuDlg_ProcessChar(stOutputValue, stVariableValue, iCaretPosition, iSelectionStart, iSelectionEnd, (flags AND VisuElems.Visu_InputFlags.Password) = 1, ';'); }
    Button (384,251 34x34), ".", invisible if: NOT bShift
        OnMouseDown: execute { VisuDlg_ProcessChar(stOutputValue, stVariableValue, iCaretPosition, iSelectionStart, iSelectionEnd, (flags AND VisuElems.Visu_InputFlags.Password) = 1, '.'); }
    Button (384,251 34x34), ":", invisible if: bShift
        OnMouseDown: execute { VisuDlg_ProcessChar(stOutputValue, stVariableValue, iCaretPosition, iSelectionStart, iSelectionEnd, (flags AND VisuElems.Visu_InputFlags.Password) = 1, ':'); }
    Button (420,251 34x34), "-", invisible if: NOT bShift
        OnMouseDown: execute { VisuDlg_ProcessChar(stOutputValue, stVariableValue, iCaretPosition, iSelectionStart, iSelectionEnd, (flags AND VisuElems.Visu_InputFlags.Password) = 1, '-'); }
    Button (420,251 34x34), "_", invisible if: bShift
        OnMouseDown: execute { VisuDlg_ProcessChar(stOutputValue, stVariableValue, iCaretPosition, iSelectionStart, iSelectionEnd, (flags AND VisuElems.Visu_InputFlags.Password) = 1, '_'); }
    Button (38,212 34x34), "€"
        OnMouseDown: execute { VisuDlg_ProcessChar(stOutputValue, stVariableValue, iCaretPosition, iSelectionStart, iSelectionEnd, (flags AND VisuElems.Visu_InputFlags.Password) = 1, '€'); }
    Button (74,212 34x34), "a", invisible if: NOT bShift
        OnMouseDown: execute { VisuDlg_ProcessChar(stOutputValue, stVariableValue, iCaretPosition, iSelectionStart, iSelectionEnd, (flags AND VisuElems.Visu_InputFlags.Password) = 1, 'a'); }
    Button (74,212 34x34), "A", invisible if: bShift
        OnMouseDown: execute { VisuDlg_ProcessChar(stOutputValue, stVariableValue, iCaretPosition, iSelectionStart, iSelectionEnd, (flags AND VisuElems.Visu_InputFlags.Password) = 1, 'A'); }
    Button (110,212 34x34), "s", invisible if: NOT bShift
        OnMouseDown: execute { VisuDlg_ProcessChar(stOutputValue, stVariableValue, iCaretPosition, iSelectionStart, iSelectionEnd, (flags AND VisuElems.Visu_InputFlags.Password) = 1, 's'); }
    Button (110,212 34x34), "S", invisible if: bShift
        OnMouseDown: execute { VisuDlg_ProcessChar(stOutputValue, stVariableValue, iCaretPosition, iSelectionStart, iSelectionEnd, (flags AND VisuElems.Visu_InputFlags.Password) = 1, 'S'); }
    Button (146,212 34x34), "d", invisible if: NOT bShift
        OnMouseDown: execute { VisuDlg_ProcessChar(stOutputValue, stVariableValue, iCaretPosition, iSelectionStart, iSelectionEnd, (flags AND VisuElems.Visu_InputFlags.Password) = 1, 'd'); }
    Button (146,212 34x34), "D", invisible if: bShift
        OnMouseDown: execute { VisuDlg_ProcessChar(stOutputValue, stVariableValue, iCaretPosition, iSelectionStart, iSelectionEnd, (flags AND VisuElems.Visu_InputFlags.Password) = 1, 'D'); }
    Button (182,212 34x34), "f", invisible if: NOT bShift
        OnMouseDown: execute { VisuDlg_ProcessChar(stOutputValue, stVariableValue, iCaretPosition, iSelectionStart, iSelectionEnd, (flags AND VisuElems.Visu_InputFlags.Password) = 1, 'f'); }
    Button (182,212 34x34), "F", invisible if: bShift
        OnMouseDown: execute { VisuDlg_ProcessChar(stOutputValue, stVariableValue, iCaretPosition, iSelectionStart, iSelectionEnd, (flags AND VisuElems.Visu_InputFlags.Password) = 1, 'F'); }
    Button (218,212 34x34), "g", invisible if: NOT bShift
        OnMouseDown: execute { VisuDlg_ProcessChar(stOutputValue, stVariableValue, iCaretPosition, iSelectionStart, iSelectionEnd, (flags AND VisuElems.Visu_InputFlags.Password) = 1, 'g'); }
    Button (218,212 34x34), "G", invisible if: bShift
        OnMouseDown: execute { VisuDlg_ProcessChar(stOutputValue, stVariableValue, iCaretPosition, iSelectionStart, iSelectionEnd, (flags AND VisuElems.Visu_InputFlags.Password) = 1, 'G'); }
    Button (254,212 34x34), "h", invisible if: NOT bShift
        OnMouseDown: execute { VisuDlg_ProcessChar(stOutputValue, stVariableValue, iCaretPosition, iSelectionStart, iSelectionEnd, (flags AND VisuElems.Visu_InputFlags.Password) = 1, 'h'); }
    Button (254,212 34x34), "H", invisible if: bShift
        OnMouseDown: execute { VisuDlg_ProcessChar(stOutputValue, stVariableValue, iCaretPosition, iSelectionStart, iSelectionEnd, (flags AND VisuElems.Visu_InputFlags.Password) = 1, 'H'); }
    Button (290,212 34x34), "j", invisible if: NOT bShift
        OnMouseDown: execute { VisuDlg_ProcessChar(stOutputValue, stVariableValue, iCaretPosition, iSelectionStart, iSelectionEnd, (flags AND VisuElems.Visu_InputFlags.Password) = 1, 'j'); }
    Button (290,212 34x34), "J", invisible if: bShift
        OnMouseDown: execute { VisuDlg_ProcessChar(stOutputValue, stVariableValue, iCaretPosition, iSelectionStart, iSelectionEnd, (flags AND VisuElems.Visu_InputFlags.Password) = 1, 'J'); }
    Button (326,212 34x34), "k", invisible if: NOT bShift
        OnMouseDown: execute { VisuDlg_ProcessChar(stOutputValue, stVariableValue, iCaretPosition, iSelectionStart, iSelectionEnd, (flags AND VisuElems.Visu_InputFlags.Password) = 1, 'k'); }
    Button (326,212 34x34), "K", invisible if: bShift
        OnMouseDown: execute { VisuDlg_ProcessChar(stOutputValue, stVariableValue, iCaretPosition, iSelectionStart, iSelectionEnd, (flags AND VisuElems.Visu_InputFlags.Password) = 1, 'K'); }
    Button (362,212 34x34), "l", invisible if: NOT bShift
        OnMouseDown: execute { VisuDlg_ProcessChar(stOutputValue, stVariableValue, iCaretPosition, iSelectionStart, iSelectionEnd, (flags AND VisuElems.Visu_InputFlags.Password) = 1, 'l'); }
    Button (362,212 34x34), "L", invisible if: bShift
        OnMouseDown: execute { VisuDlg_ProcessChar(stOutputValue, stVariableValue, iCaretPosition, iSelectionStart, iSelectionEnd, (flags AND VisuElems.Visu_InputFlags.Password) = 1, 'L'); }
    Button (398,212 34x34), "ö", invisible if: NOT bShift
        OnMouseDown: execute { VisuDlg_ProcessChar(stOutputValue, stVariableValue, iCaretPosition, iSelectionStart, iSelectionEnd, (flags AND VisuElems.Visu_InputFlags.Password) = 1, 'ö'); }
    Button (398,212 34x34), "Ö", invisible if: bShift
        OnMouseDown: execute { VisuDlg_ProcessChar(stOutputValue, stVariableValue, iCaretPosition, iSelectionStart, iSelectionEnd, (flags AND VisuElems.Visu_InputFlags.Password) = 1, 'Ö'); }
    Button (434,212 34x34), "ä", invisible if: NOT bShift
        OnMouseDown: execute { VisuDlg_ProcessChar(stOutputValue, stVariableValue, iCaretPosition, iSelectionStart, iSelectionEnd, (flags AND VisuElems.Visu_InputFlags.Password) = 1, 'ä'); }
    Button (434,212 34x34), "Ä", invisible if: bShift
        OnMouseDown: execute { VisuDlg_ProcessChar(stOutputValue, stVariableValue, iCaretPosition, iSelectionStart, iSelectionEnd, (flags AND VisuElems.Visu_InputFlags.Password) = 1, 'Ä'); }
    Button (470,212 34x34), "#", invisible if: NOT bShift
        OnMouseDown: execute { VisuDlg_ProcessChar(stOutputValue, stVariableValue, iCaretPosition, iSelectionStart, iSelectionEnd, (flags AND VisuElems.Visu_InputFlags.Password) = 1, '#'); }
    Button (470,212 34x34), "'", invisible if: bShift
        OnMouseDown: execute { VisuDlg_ProcessChar(stOutputValue, stVariableValue, iCaretPosition, iSelectionStart, iSelectionEnd, (flags AND VisuElems.Visu_InputFlags.Password) = 1, '$''); }
    Button (24,173 34x34), "@"
        OnMouseDown: execute { VisuDlg_ProcessChar(stOutputValue, stVariableValue, iCaretPosition, iSelectionStart, iSelectionEnd, (flags AND VisuElems.Visu_InputFlags.Password) = 1, '@'); }
    Button (60,173 34x34), "q", invisible if: NOT bShift
        OnMouseDown: execute { VisuDlg_ProcessChar(stOutputValue, stVariableValue, iCaretPosition, iSelectionStart, iSelectionEnd, (flags AND VisuElems.Visu_InputFlags.Password) = 1, 'q'); }
    Button (60,173 34x34), "Q", invisible if: bShift
        OnMouseDown: execute { VisuDlg_ProcessChar(stOutputValue, stVariableValue, iCaretPosition, iSelectionStart, iSelectionEnd, (flags AND VisuElems.Visu_InputFlags.Password) = 1, 'Q'); }
    Button (96,173 34x34), "w", invisible if: NOT bShift
        OnMouseDown: execute { VisuDlg_ProcessChar(stOutputValue, stVariableValue, iCaretPosition, iSelectionStart, iSelectionEnd, (flags AND VisuElems.Visu_InputFlags.Password) = 1, 'w'); }
    Button (96,173 34x34), "W", invisible if: bShift
        OnMouseDown: execute { VisuDlg_ProcessChar(stOutputValue, stVariableValue, iCaretPosition, iSelectionStart, iSelectionEnd, (flags AND VisuElems.Visu_InputFlags.Password) = 1, 'W'); }
    Button (132,173 34x34), "e", invisible if: NOT bShift
        OnMouseDown: execute { VisuDlg_ProcessChar(stOutputValue, stVariableValue, iCaretPosition, iSelectionStart, iSelectionEnd, (flags AND VisuElems.Visu_InputFlags.Password) = 1, 'e'); }
    Button (132,173 34x34), "E", invisible if: bShift
        OnMouseDown: execute { VisuDlg_ProcessChar(stOutputValue, stVariableValue, iCaretPosition, iSelectionStart, iSelectionEnd, (flags AND VisuElems.Visu_InputFlags.Password) = 1, 'E'); }
    Button (168,173 34x34), "r", invisible if: NOT bShift
        OnMouseDown: execute { VisuDlg_ProcessChar(stOutputValue, stVariableValue, iCaretPosition, iSelectionStart, iSelectionEnd, (flags AND VisuElems.Visu_InputFlags.Password) = 1, 'r'); }
    Button (168,173 34x34), "R", invisible if: bShift
        OnMouseDown: execute { VisuDlg_ProcessChar(stOutputValue, stVariableValue, iCaretPosition, iSelectionStart, iSelectionEnd, (flags AND VisuElems.Visu_InputFlags.Password) = 1, 'R'); }
    Button (204,173 34x34), "t", invisible if: NOT bShift
        OnMouseDown: execute { VisuDlg_ProcessChar(stOutputValue, stVariableValue, iCaretPosition, iSelectionStart, iSelectionEnd, (flags AND VisuElems.Visu_InputFlags.Password) = 1, 't'); }
    Button (204,173 34x34), "T", invisible if: bShift
        OnMouseDown: execute { VisuDlg_ProcessChar(stOutputValue, stVariableValue, iCaretPosition, iSelectionStart, iSelectionEnd, (flags AND VisuElems.Visu_InputFlags.Password) = 1, 'T'); }
    Button (240,173 34x34), "z", invisible if: NOT bShift
        OnMouseDown: execute { VisuDlg_ProcessChar(stOutputValue, stVariableValue, iCaretPosition, iSelectionStart, iSelectionEnd, (flags AND VisuElems.Visu_InputFlags.Password) = 1, 'z'); }
    Button (240,173 34x34), "Z", invisible if: bShift
        OnMouseDown: execute { VisuDlg_ProcessChar(stOutputValue, stVariableValue, iCaretPosition, iSelectionStart, iSelectionEnd, (flags AND VisuElems.Visu_InputFlags.Password) = 1, 'Z'); }
    Button (276,173 34x34), "u", invisible if: NOT bShift
        OnMouseDown: execute { VisuDlg_ProcessChar(stOutputValue, stVariableValue, iCaretPosition, iSelectionStart, iSelectionEnd, (flags AND VisuElems.Visu_InputFlags.Password) = 1, 'u'); }
    Button (276,173 34x34), "U", invisible if: bShift
        OnMouseDown: execute { VisuDlg_ProcessChar(stOutputValue, stVariableValue, iCaretPosition, iSelectionStart, iSelectionEnd, (flags AND VisuElems.Visu_InputFlags.Password) = 1, 'U'); }
    Button (312,173 34x34), "i", invisible if: NOT bShift
        OnMouseDown: execute { VisuDlg_ProcessChar(stOutputValue, stVariableValue, iCaretPosition, iSelectionStart, iSelectionEnd, (flags AND VisuElems.Visu_InputFlags.Password) = 1, 'i'); }
    Button (312,173 34x34), "I", invisible if: bShift
        OnMouseDown: execute { VisuDlg_ProcessChar(stOutputValue, stVariableValue, iCaretPosition, iSelectionStart, iSelectionEnd, (flags AND VisuElems.Visu_InputFlags.Password) = 1, 'I'); }
    Button (348,173 34x34), "o", invisible if: NOT bShift
        OnMouseDown: execute { VisuDlg_ProcessChar(stOutputValue, stVariableValue, iCaretPosition, iSelectionStart, iSelectionEnd, (flags AND VisuElems.Visu_InputFlags.Password) = 1, 'o'); }
    Button (348,173 34x34), "O", invisible if: bShift
        OnMouseDown: execute { VisuDlg_ProcessChar(stOutputValue, stVariableValue, iCaretPosition, iSelectionStart, iSelectionEnd, (flags AND VisuElems.Visu_InputFlags.Password) = 1, 'O'); }
    Button (384,173 34x34), "p", invisible if: NOT bShift
        OnMouseDown: execute { VisuDlg_ProcessChar(stOutputValue, stVariableValue, iCaretPosition, iSelectionStart, iSelectionEnd, (flags AND VisuElems.Visu_InputFlags.Password) = 1, 'p'); }
    Button (384,173 34x34), "P", invisible if: bShift
        OnMouseDown: execute { VisuDlg_ProcessChar(stOutputValue, stVariableValue, iCaretPosition, iSelectionStart, iSelectionEnd, (flags AND VisuElems.Visu_InputFlags.Password) = 1, 'P'); }
    Button (420,173 34x34), "ü", invisible if: NOT bShift
        OnMouseDown: execute { VisuDlg_ProcessChar(stOutputValue, stVariableValue, iCaretPosition, iSelectionStart, iSelectionEnd, (flags AND VisuElems.Visu_InputFlags.Password) = 1, 'ü'); }
    Button (420,173 34x34), "Ü", invisible if: bShift
        OnMouseDown: execute { VisuDlg_ProcessChar(stOutputValue, stVariableValue, iCaretPosition, iSelectionStart, iSelectionEnd, (flags AND VisuElems.Visu_InputFlags.Password) = 1, 'Ü'); }
    Button (456,173 34x34), "+", invisible if: NOT bShift
        OnMouseDown: execute { VisuDlg_ProcessChar(stOutputValue, stVariableValue, iCaretPosition, iSelectionStart, iSelectionEnd, (flags AND VisuElems.Visu_InputFlags.Password) = 1, '+'); }
    Button (456,173 34x34), "*", invisible if: bShift
        OnMouseDown: execute { VisuDlg_ProcessChar(stOutputValue, stVariableValue, iCaretPosition, iSelectionStart, iSelectionEnd, (flags AND VisuElems.Visu_InputFlags.Password) = 1, '*'); }
    Button (492,173 34x34), "~"
        OnMouseDown: execute { VisuDlg_ProcessChar(stOutputValue, stVariableValue, iCaretPosition, iSelectionStart, iSelectionEnd, (flags AND VisuElems.Visu_InputFlags.Password) = 1, '~'); }
    Button (11,135 34x34), "^", invisible if: NOT bShift
        OnMouseDown: execute { VisuDlg_ProcessChar(stOutputValue, stVariableValue, iCaretPosition, iSelectionStart, iSelectionEnd, (flags AND VisuElems.Visu_InputFlags.Password) = 1, '^'); }
    Button (11,135 34x34), "°", invisible if: bShift
        OnMouseDown: execute { VisuDlg_ProcessChar(stOutputValue, stVariableValue, iCaretPosition, iSelectionStart, iSelectionEnd, (flags AND VisuElems.Visu_InputFlags.Password) = 1, '°'); }
    Button (47,135 34x34), "1", invisible if: NOT bShift
        OnMouseDown: execute { VisuDlg_ProcessChar(stOutputValue, stVariableValue, iCaretPosition, iSelectionStart, iSelectionEnd, (flags AND VisuElems.Visu_InputFlags.Password) = 1, '1'); }
    Button (47,135 34x34), "!", invisible if: bShift
        OnMouseDown: execute { VisuDlg_ProcessChar(stOutputValue, stVariableValue, iCaretPosition, iSelectionStart, iSelectionEnd, (flags AND VisuElems.Visu_InputFlags.Password) = 1, '!'); }
    Button (83,135 34x34), "2", invisible if: NOT bShift
        OnMouseDown: execute { VisuDlg_ProcessChar(stOutputValue, stVariableValue, iCaretPosition, iSelectionStart, iSelectionEnd, (flags AND VisuElems.Visu_InputFlags.Password) = 1, '2'); }
    Button (83,135 34x34), """, invisible if: bShift
        OnMouseDown: execute { VisuDlg_ProcessChar(stOutputValue, stVariableValue, iCaretPosition, iSelectionStart, iSelectionEnd, (flags AND VisuElems.Visu_InputFlags.Password) = 1, '"'); }
    Button (119,135 34x34), "3", invisible if: NOT bShift
        OnMouseDown: execute { VisuDlg_ProcessChar(stOutputValue, stVariableValue, iCaretPosition, iSelectionStart, iSelectionEnd, (flags AND VisuElems.Visu_InputFlags.Password) = 1, '3'); }
    Button (119,135 34x34), "§", invisible if: bShift
        OnMouseDown: execute { VisuDlg_ProcessChar(stOutputValue, stVariableValue, iCaretPosition, iSelectionStart, iSelectionEnd, (flags AND VisuElems.Visu_InputFlags.Password) = 1, '§'); }
    Button (155,135 34x34), "4", invisible if: NOT bShift
        OnMouseDown: execute { VisuDlg_ProcessChar(stOutputValue, stVariableValue, iCaretPosition, iSelectionStart, iSelectionEnd, (flags AND VisuElems.Visu_InputFlags.Password) = 1, '4'); }
    Button (155,135 34x34), "$", invisible if: bShift
        OnMouseDown: execute { VisuDlg_ProcessChar(stOutputValue, stVariableValue, iCaretPosition, iSelectionStart, iSelectionEnd, (flags AND VisuElems.Visu_InputFlags.Password) = 1, '$$'); }
    Button (191,135 34x34), "5", invisible if: NOT bShift
        OnMouseDown: execute { VisuDlg_ProcessChar(stOutputValue, stVariableValue, iCaretPosition, iSelectionStart, iSelectionEnd, (flags AND VisuElems.Visu_InputFlags.Password) = 1, '5'); }
    Button (191,135 34x34), "%", invisible if: bShift
        OnMouseDown: execute { VisuDlg_ProcessChar(stOutputValue, stVariableValue, iCaretPosition, iSelectionStart, iSelectionEnd, (flags AND VisuElems.Visu_InputFlags.Password) = 1, '%'); }
    Button (227,135 34x34), "6", invisible if: NOT bShift
        OnMouseDown: execute { VisuDlg_ProcessChar(stOutputValue, stVariableValue, iCaretPosition, iSelectionStart, iSelectionEnd, (flags AND VisuElems.Visu_InputFlags.Password) = 1, '6'); }
    Button (227,135 34x34), "&", invisible if: bShift
        OnMouseDown: execute { VisuDlg_ProcessChar(stOutputValue, stVariableValue, iCaretPosition, iSelectionStart, iSelectionEnd, (flags AND VisuElems.Visu_InputFlags.Password) = 1, '&'); }
    Button (263,135 34x34), "7", invisible if: NOT bShift
        OnMouseDown: execute { VisuDlg_ProcessChar(stOutputValue, stVariableValue, iCaretPosition, iSelectionStart, iSelectionEnd, (flags AND VisuElems.Visu_InputFlags.Password) = 1, '7'); }
    Button (263,135 34x34), "/", invisible if: bShift
        OnMouseDown: execute { VisuDlg_ProcessChar(stOutputValue, stVariableValue, iCaretPosition, iSelectionStart, iSelectionEnd, (flags AND VisuElems.Visu_InputFlags.Password) = 1, '/'); }
    Button (299,135 34x34), "8", invisible if: NOT bShift
        OnMouseDown: execute { VisuDlg_ProcessChar(stOutputValue, stVariableValue, iCaretPosition, iSelectionStart, iSelectionEnd, (flags AND VisuElems.Visu_InputFlags.Password) = 1, '8'); }
    Button (299,135 34x34), "(", invisible if: bShift
        OnMouseDown: execute { VisuDlg_ProcessChar(stOutputValue, stVariableValue, iCaretPosition, iSelectionStart, iSelectionEnd, (flags AND VisuElems.Visu_InputFlags.Password) = 1, '('); }
    Button (335,135 34x34), "9", invisible if: NOT bShift
        OnMouseDown: execute { VisuDlg_ProcessChar(stOutputValue, stVariableValue, iCaretPosition, iSelectionStart, iSelectionEnd, (flags AND VisuElems.Visu_InputFlags.Password) = 1, '9'); }
    Button (335,135 34x34), ")", invisible if: bShift
        OnMouseDown: execute { VisuDlg_ProcessChar(stOutputValue, stVariableValue, iCaretPosition, iSelectionStart, iSelectionEnd, (flags AND VisuElems.Visu_InputFlags.Password) = 1, ')'); }
    Button (371,135 34x34), "0", invisible if: NOT bShift
        OnMouseDown: execute { VisuDlg_ProcessChar(stOutputValue, stVariableValue, iCaretPosition, iSelectionStart, iSelectionEnd, (flags AND VisuElems.Visu_InputFlags.Password) = 1, '0'); }
    Button (371,135 34x34), "=", invisible if: bShift
        OnMouseDown: execute { VisuDlg_ProcessChar(stOutputValue, stVariableValue, iCaretPosition, iSelectionStart, iSelectionEnd, (flags AND VisuElems.Visu_InputFlags.Password) = 1, '='); }
    Button (407,135 34x34), "ß", invisible if: NOT bShift
        OnMouseDown: execute { VisuDlg_ProcessChar(stOutputValue, stVariableValue, iCaretPosition, iSelectionStart, iSelectionEnd, (flags AND VisuElems.Visu_InputFlags.Password) = 1, 'ß'); }
    Button (407,135 34x34), "?", invisible if: bShift
        OnMouseDown: execute { VisuDlg_ProcessChar(stOutputValue, stVariableValue, iCaretPosition, iSelectionStart, iSelectionEnd, (flags AND VisuElems.Visu_InputFlags.Password) = 1, '?'); }
    Button (443,135 34x34), "´"
        OnMouseDown: execute { VisuDlg_ProcessChar(stOutputValue, stVariableValue, iCaretPosition, iSelectionStart, iSelectionEnd, (flags AND VisuElems.Visu_InputFlags.Password) = 1, '´'); }
    Button (479,135 34x34), "\"
        OnMouseDown: execute { VisuDlg_ProcessChar(stOutputValue, stVariableValue, iCaretPosition, iSelectionStart, iSelectionEnd, (flags AND VisuElems.Visu_InputFlags.Password) = 1, '\'); }
    Rectangle (2,67 578x62)
    Rectangle (21,105 546x20), "%s", text variable: stMessage
    Rectangle (578,2 3x332)
    Rectangle (1,2 3x332)
    Rectangle (1,333 580x4)
    Polyline (16,128) (16,101) (568,101)
    Polyline (16,96) (16,69) (568,69)
    Polyline (17,128) (568,128) (568,101)
    Polyline (17,96) (568,96) (568,69)
    Image (1,2 580x29), image: Title2
    Rectangle (1,2 579x28), invisible if: VisuElems.g_VisualizationStyle.GetDINT('Dialog-UseHeaderColor', 0, 0) = 0
    Rectangle (12,7 563x20), "%s", text variable: wstTitle
    Rectangle (21,72 31x20), "Min:", invisible if: LEN(stMin) = 0
        p55702900: SEL(((UDINT_TO_DINT(flags AND 16#008))=16#0010),16#FF000000,16#FFFF0000)
    Rectangle (50,72 95x20), "%s", text variable: stMin, invisible if: LEN(stMin) = 0
        p55702900: SEL(((UDINT_TO_DINT(flags AND 16#0010))=16#0010),16#FF000000,16#FFFF0000)
    Rectangle (208,72 31x20), "Max:", invisible if: LEN(stMax) = 0
        p55702900: SEL(((UDINT_TO_DINT(flags AND 16#0010))=16#0010),16#FF000000,16#FFFF0000)
    Rectangle (241,72 95x20), "%s", text variable: stMax, invisible if: LEN(stMax) = 0
        p55702900: SEL(((UDINT_TO_DINT(flags AND 16#0010))=16#0010),16#FF000000,16#FFFF0000)
END_VISUALIZATION

// ---- VISUs/Keyboard/Numpad.TcVIS
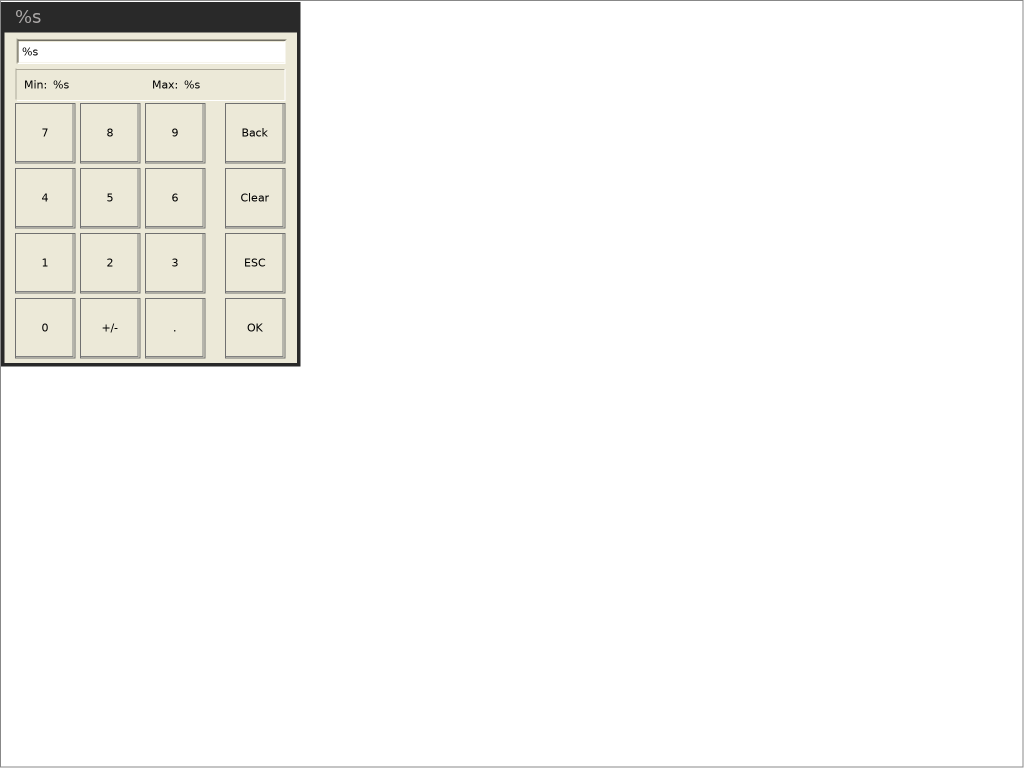
VISUALIZATION Numpad  // 1024x768
VAR_INPUT
	stVariableValue : STRING;
	stMin : STRING;
	stMax : STRING;
	wstTitle : WSTRING;
	flags : DWORD;
END_VAR
VAR
	bInit : BOOL;
	stMessage : STRING;
	stOutputValue : STRING;
	iCaretPosition	: INT;
	iSelectionStart	: INT;
	iSelectionEnd	: INT;
	xAllSelected	: BOOL;
END_VAR
    Rectangle (3,31 294x39)
    Polyline (17,63) (17,39) (286,39)
    Polyline (18,63) (285,63) (285,40)
    Polyline (18,62) (18,40) (285,40)
    Textfield (19,42 265x20), "%s", text variable: stOutputValue
        p905179711: iCaretPosition
        p3815007873: iSelectionStart
        p1425650380: iSelectionEnd
        p3479897389: xAllSelected
    Rectangle (3,98 295x67)
    Rectangle (3,165 295x65)
    Rectangle (3,230 295x65)
    Rectangle (3,295 295x68)
    Button (225,298 60x60), "OK"
        OnMouseDown: CloseDialog Dialog=Numpad, Result=OK, NumpadKeypad=True, NumpadKeypadSet=True
    Button (225,233 60x60), "ESC"
        OnMouseDown: CloseDialog Dialog=Numpad, Result=Cancel, NumpadKeypad=True, NumpadKeypadSet=True
    Button (225,168 60x60), "Clear"
        OnMouseDown: execute {
            stVariableValue := '';
            stOutputValue := '';
            flags := flags AND NOT 16#0008;
            flags := flags AND NOT 16#0010;
            iCaretPosition	:= 1;
            iSelectionStart	:= 1;
            iSelectionEnd	:= 1;
        }
    Button (225,103 60x60), "Back"
        OnMouseDown: execute { VisuDlg_ProcessBack(stOutputValue, stVariableValue, iCaretPosition, iSelectionStart, iSelectionEnd, bInit); }
    Button (145,298 60x60), "."
        OnMouseDown: execute { VisuDlg_ProcessChar(stOutputValue, stVariableValue, iCaretPosition, iSelectionStart, iSelectionEnd, (flags AND VisuElems.Visu_InputFlags.Password) = 1, '.'); }
    Button (80,298 60x60), "+/-"
        OnMouseDown: execute { VisuDlg_ProcessChangeSign(stOutputValue, stVariableValue, iCaretPosition, iSelectionStart, iSelectionEnd, (flags AND VisuElems.Visu_InputFlags.Password) = 1); }
    Button (15,298 60x60), "0"
        OnMouseDown: execute { VisuDlg_ProcessChar(stOutputValue, stVariableValue, iCaretPosition, iSelectionStart, iSelectionEnd, (flags AND VisuElems.Visu_InputFlags.Password) = 1, '0'); }
    Button (15,233 60x60), "1"
        OnMouseDown: execute { VisuDlg_ProcessChar(stOutputValue, stVariableValue, iCaretPosition, iSelectionStart, iSelectionEnd, (flags AND VisuElems.Visu_InputFlags.Password) = 1, '1'); }
    Button (80,233 60x60), "2"
        OnMouseDown: execute { VisuDlg_ProcessChar(stOutputValue, stVariableValue, iCaretPosition, iSelectionStart, iSelectionEnd, (flags AND VisuElems.Visu_InputFlags.Password) = 1, '2'); }
    Button (145,233 60x60), "3"
        OnMouseDown: execute { VisuDlg_ProcessChar(stOutputValue, stVariableValue, iCaretPosition, iSelectionStart, iSelectionEnd, (flags AND VisuElems.Visu_InputFlags.Password) = 1, '3'); }
    Button (15,168 60x60), "4"
        OnMouseDown: execute { VisuDlg_ProcessChar(stOutputValue, stVariableValue, iCaretPosition, iSelectionStart, iSelectionEnd, (flags AND VisuElems.Visu_InputFlags.Password) = 1, '4'); }
    Button (80,168 60x60), "5"
        OnMouseDown: execute { VisuDlg_ProcessChar(stOutputValue, stVariableValue, iCaretPosition, iSelectionStart, iSelectionEnd, (flags AND VisuElems.Visu_InputFlags.Password) = 1, '5'); }
    Button (145,168 60x60), "6"
        OnMouseDown: execute { VisuDlg_ProcessChar(stOutputValue, stVariableValue, iCaretPosition, iSelectionStart, iSelectionEnd, (flags AND VisuElems.Visu_InputFlags.Password) = 1, '6'); }
    Button (15,103 60x60), "7"
        OnMouseDown: execute { VisuDlg_ProcessChar(stOutputValue, stVariableValue, iCaretPosition, iSelectionStart, iSelectionEnd, (flags AND VisuElems.Visu_InputFlags.Password) = 1, '7'); }
    Button (80,103 60x60), "8"
        OnMouseDown: execute { VisuDlg_ProcessChar(stOutputValue, stVariableValue, iCaretPosition, iSelectionStart, iSelectionEnd, (flags AND VisuElems.Visu_InputFlags.Password) = 1, '8'); }
    Button (145,103 60x60), "9"
        OnMouseDown: execute { VisuDlg_ProcessChar(stOutputValue, stVariableValue, iCaretPosition, iSelectionStart, iSelectionEnd, (flags AND VisuElems.Visu_InputFlags.Password) = 1, '9'); }
    Rectangle (3,69 294x33)
    Rectangle (50,75 95x20), "%s", text variable: stMin, invisible if: LEN(stMin) = 0
        p55702900: SEL(((UDINT_TO_DINT(flags AND 16#0008))=16#0008),16#FF000000,16#FFFF0000)
    Rectangle (181,75 95x20), "%s", text variable: stMax, invisible if: LEN(stMax) = 0
        p55702900: SEL(((UDINT_TO_DINT(flags AND 16#0010))=16#0010),16#FF000000,16#FFFF0000)
    Rectangle (149,75 31x20), "Max:", invisible if: LEN(stMax) = 0
        p55702900: SEL(((UDINT_TO_DINT(flags AND 16#0010))=16#0010),16#FF000000,16#FFFF0000)
    Rectangle (296,363 3x3)
    Rectangle (297,2 3x362)
    Rectangle (1,3 3x360)
    Rectangle (1,2 298x30), invisible if: VisuElems.g_VisualizationStyle.GetDINT('Dialog-UseHeaderColor', 0, 0) = 0
    Rectangle (12,7 280x20), "%s", text variable: gsPadTitle
    Rectangle (1,363 299x3)
    Polyline (16,99) (16,69) (284,69)
    Polyline (17,100) (285,100) (285,69)
    Rectangle (21,75 31x20), "Min:", invisible if: LEN(stMin) = 0
        p55702900: SEL(((UDINT_TO_DINT(flags AND 16#0008))=16#0008),16#FF000000,16#FFFF0000)
END_VISUALIZATION

// ---- VISUs/Keyboard/NumpadExtended.TcVIS
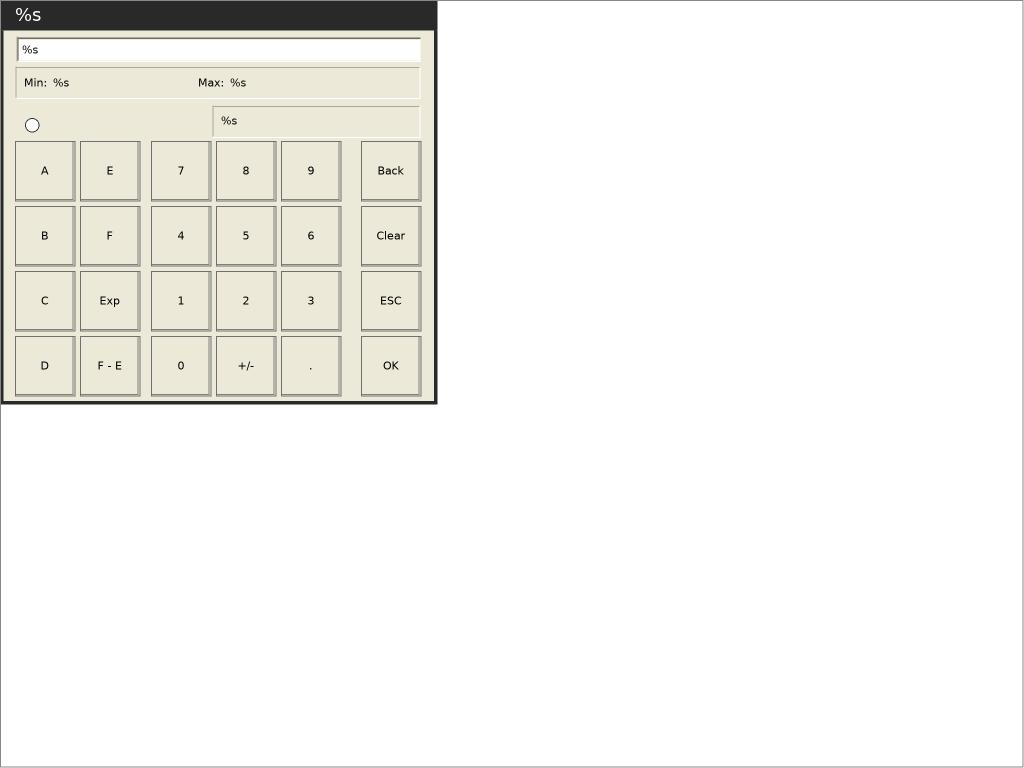
VISUALIZATION NumpadExtended  // 1024x768
VAR_INPUT
	stVariableValue : STRING;
	stMin : STRING;
	stMax : STRING;
	wstTitle : WSTRING;
	flags : DWORD;	
END_VAR
VAR
	bInit : BOOL;
	stMessage : STRING;
	// the display value
	stOutputValue : STRING;		
	// 0: dec, 1: hex, like Dialog_FormatTypes
	iFormatValue : INT;
	bInitFormatValue : BOOL;	
	iCaretPosition	: INT;
	iSelectionStart	: INT;
	iSelectionEnd	: INT;
	xAllSelected	: BOOL;
END_VAR
    Rectangle (3,29 434x39)
    Polyline (17,61) (17,37) (420,37)
    Polyline (18,61) (420,61) (420,38)
    Polyline (18,60) (18,38) (420,38)
    Textfield (19,40 400x20), "%s", text variable: stOutputValue
        p905179711: iCaretPosition
        p3815007873: iSelectionStart
        p1425650380: iSelectionEnd
        p3479897389: xAllSelected
    Rectangle (3,136 434x266)
    Button (361,336 60x60), "OK"
        OnMouseDown: execute { VisuDlgUtil_CloseNumpadExtended2(stOutputValue, stVariableValue, stMin, stMax, iFormatValue, bInitFormatValue, iCaretPosition, iSelectionStart, iSelectionEnd, flags); }
        OnMouseDown: CloseDialog Dialog=NumpadExtended, Result=OK, NumpadKeypad=True, NumpadKeypadSet=True
    Button (361,271 60x60), "ESC"
        OnMouseDown: execute { VisuDlgUtil_SetbInitFormatValue(bInitFormatValue, '0'); }
        OnMouseDown: CloseDialog Dialog=NumpadExtended, Result=Cancel, NumpadKeypad=True, NumpadKeypadSet=True
    Button (361,206 60x60), "Clear"
        OnMouseDown: execute { VisuDlg_ProcessClear(stOutputValue, stVariableValue, flags, iCaretPosition, iSelectionStart, iSelectionEnd); }
    Button (361,141 60x60), "Back"
        OnMouseDown: execute { VisuDlg_ProcessBack(stOutputValue, stVariableValue, iCaretPosition, iSelectionStart, iSelectionEnd, bInit); }
    Button (281,336 60x60), ".", input disabled if: iFormatValue = 1
        OnMouseDown: execute { VisuDlg_ProcessCharWithInit(stOutputValue, stVariableValue, iCaretPosition, iSelectionStart, iSelectionEnd, bInit, (flags AND VisuElems.Visu_InputFlags.Password) = 1, '.'); }
    Button (216,336 60x60), "+/-"
        OnMouseDown: execute { VisuDlg_ProcessChangeSignExtended(stOutputValue, stVariableValue, iCaretPosition, iSelectionStart, iSelectionEnd, bInit, (flags AND VisuElems.Visu_InputFlags.Password) = 1, iFormatValue); }
    Button (151,336 60x60), "0"
        OnMouseDown: execute { VisuDlg_ProcessCharWithInit(stOutputValue, stVariableValue, iCaretPosition, iSelectionStart, iSelectionEnd, bInit, (flags AND VisuElems.Visu_InputFlags.Password) = 1, '0'); }
    Button (151,271 60x60), "1"
        OnMouseDown: execute { VisuDlg_ProcessCharWithInit(stOutputValue, stVariableValue, iCaretPosition, iSelectionStart, iSelectionEnd, bInit, (flags AND VisuElems.Visu_InputFlags.Password) = 1, '1'); }
    Button (216,271 60x60), "2"
        OnMouseDown: execute { VisuDlg_ProcessCharWithInit(stOutputValue, stVariableValue, iCaretPosition, iSelectionStart, iSelectionEnd, bInit, (flags AND VisuElems.Visu_InputFlags.Password) = 1, '2'); }
    Button (281,271 60x60), "3"
        OnMouseDown: execute { VisuDlg_ProcessCharWithInit(stOutputValue, stVariableValue, iCaretPosition, iSelectionStart, iSelectionEnd, bInit, (flags AND VisuElems.Visu_InputFlags.Password) = 1, '3'); }
    Button (151,206 60x60), "4"
        OnMouseDown: execute { VisuDlg_ProcessCharWithInit(stOutputValue, stVariableValue, iCaretPosition, iSelectionStart, iSelectionEnd, bInit, (flags AND VisuElems.Visu_InputFlags.Password) = 1, '4'); }
    Button (216,206 60x60), "5"
        OnMouseDown: execute { VisuDlg_ProcessCharWithInit(stOutputValue, stVariableValue, iCaretPosition, iSelectionStart, iSelectionEnd, bInit, (flags AND VisuElems.Visu_InputFlags.Password) = 1, '5'); }
    Button (281,206 60x60), "6"
        OnMouseDown: execute { VisuDlg_ProcessCharWithInit(stOutputValue, stVariableValue, iCaretPosition, iSelectionStart, iSelectionEnd, bInit, (flags AND VisuElems.Visu_InputFlags.Password) = 1, '6'); }
    Button (151,141 60x60), "7"
        OnMouseDown: execute { VisuDlg_ProcessCharWithInit(stOutputValue, stVariableValue, iCaretPosition, iSelectionStart, iSelectionEnd, bInit, (flags AND VisuElems.Visu_InputFlags.Password) = 1, '7'); }
    Button (216,141 60x60), "8"
        OnMouseDown: execute { VisuDlg_ProcessCharWithInit(stOutputValue, stVariableValue, iCaretPosition, iSelectionStart, iSelectionEnd, bInit, (flags AND VisuElems.Visu_InputFlags.Password) = 1, '8'); }
    Button (281,141 60x60), "9"
        OnMouseDown: execute { VisuDlg_ProcessCharWithInit(stOutputValue, stVariableValue, iCaretPosition, iSelectionStart, iSelectionEnd, bInit, (flags AND VisuElems.Visu_InputFlags.Password) = 1, '9'); }
    Rectangle (3,67 434x69)
        p3560616238: VisuDlgUtil_InitValueFromFlags(flags, bInitFormatValue, iFormatValue)
    Rectangle (50,73 120x20), "%s", text variable: stMin, invisible if: LEN(stMin) = 0
    Rectangle (227,73 120x20), "%s", text variable: stMax, invisible if: LEN(stMax) = 0
    Rectangle (195,73 31x20), "Max:", text variable: stMin, invisible if: LEN(stMax) = 0
        p55702900: SEL(((UDINT_TO_DINT(flags AND 16#0010))=16#0010),16#FF000000,16#FFFF0000)
    Rectangle (296,401 3x3)
    Rectangle (434,0 3x404)
    Rectangle (0,0 3x404)
    Image (2,0 434x30), image: Title
    Rectangle (2,0 434x30), invisible if: VisuElems.g_VisualizationStyle.GetDINT('Dialog-UseHeaderColor', 0, 0) = 0
    Rectangle (12,5 406x20), "%s", text variable: wstTitle
    Rectangle (1,401 434x3)
    Polyline (213,136) (213,106) (419,106)
    Polyline (16,97) (16,67) (420,67)
    Polyline (213,137) (420,137) (420,106)
    Polyline (17,98) (420,98) (420,67)
    Rectangle (218,111 195x20), "%s", text variable: stMessage
    Rectangle (21,73 31x20), "Min:", text variable: stMin, invisible if: LEN(stMin) = 0
        p55702900: SEL(((UDINT_TO_DINT(flags AND 16#0008))=16#0008),16#FF000000,16#FFFF0000)
    Button (80,336 60x60), "F - E", input disabled if: iFormatValue = 1
        OnMouseDown: execute { VisuDlg_ProcessExpFloatFormatSwitch(stOutputValue, stVariableValue, iCaretPosition, iSelectionStart, iSelectionEnd, bInit, (flags AND VisuElems.Visu_InputFlags.Password) = 1); }
    Button (80,271 60x60), "Exp", input disabled if: iFormatValue = 1
        OnMouseDown: execute { VisuDlg_ProcessExp(stOutputValue, stVariableValue, iCaretPosition, iSelectionStart, iSelectionEnd, bInit, (flags AND VisuElems.Visu_InputFlags.Password) = 1); }
    Button (80,141 60x60), "E", input disabled if: iFormatValue = 0
        OnMouseDown: execute { VisuDlg_ProcessCharWithInit(stOutputValue, stVariableValue, iCaretPosition, iSelectionStart, iSelectionEnd, bInit, (flags AND VisuElems.Visu_InputFlags.Password) = 1, 'E'); }
    Button (80,206 60x60), "F", input disabled if: iFormatValue = 0
        OnMouseDown: execute { VisuDlg_ProcessCharWithInit(stOutputValue, stVariableValue, iCaretPosition, iSelectionStart, iSelectionEnd, bInit, (flags AND VisuElems.Visu_InputFlags.Password) = 1, 'F'); }
    Button (15,336 60x60), "D", input disabled if: iFormatValue = 0
        OnMouseDown: execute { VisuDlg_ProcessCharWithInit(stOutputValue, stVariableValue, iCaretPosition, iSelectionStart, iSelectionEnd, bInit, (flags AND VisuElems.Visu_InputFlags.Password) = 1, 'D'); }
    Button (15,271 60x60), "C", input disabled if: iFormatValue = 0
        OnMouseDown: execute { VisuDlg_ProcessCharWithInit(stOutputValue, stVariableValue, iCaretPosition, iSelectionStart, iSelectionEnd, bInit, (flags AND VisuElems.Visu_InputFlags.Password) = 1, 'C'); }
    Button (15,206 60x60), "B", input disabled if: iFormatValue = 0
        OnMouseDown: execute { VisuDlg_ProcessCharWithInit(stOutputValue, stVariableValue, iCaretPosition, iSelectionStart, iSelectionEnd, bInit, (flags AND VisuElems.Visu_InputFlags.Password) = 1, 'B'); }
    Button (15,141 60x60), "A", input disabled if: iFormatValue = 0
        OnMouseDown: execute { VisuDlg_ProcessCharWithInit(stOutputValue, stVariableValue, iCaretPosition, iSelectionStart, iSelectionEnd, bInit, (flags AND VisuElems.Visu_InputFlags.Password) = 1, 'A'); }
    RadioButton (23,110 150x30), variable: iFormatValue
        Areas[0]: Text=Dec
        Areas[1]: Text=Hex
    InvisibleInput (21,104 72x30)
        OnMouseDown: execute { VisuDlg_ProcessChangeNumberFormat(stOutputValue, stVariableValue, stMin, stMax, iFormatValue, iCaretPosition, iSelectionStart, iSelectionEnd, (flags AND VisuElems.Visu_InputFlags.Password) = 1, '0'); }
    InvisibleInput (96,104 72x30)
        OnMouseDown: execute { VisuDlg_ProcessChangeNumberFormat(stOutputValue, stVariableValue, stMin, stMax, iFormatValue, iCaretPosition, iSelectionStart, iSelectionEnd, (flags AND VisuElems.Visu_InputFlags.Password) = 1, '1'); }
END_VISUALIZATION

